// TwinCAT 3 PLC project HMISample
// ProgramVersion: 3.1.4022.1
// CompilerDefines: VISU_USEWSTRING
// libraries:
//   Tc2_ProfinetDiag, * (Beckhoff Automation GmbH)
//   Tc2_Standard, * (Beckhoff Automation GmbH)
//   Tc2_System, * (Beckhoff Automation GmbH)
//   Tc2_SystemCX, * (Beckhoff Automation GmbH)
//   Tc2_Utilities, * (Beckhoff Automation GmbH)
//   Tc3_Module, * (Beckhoff Automation GmbH)
//   VisuDialogs, * (System)
//   VisuSymbols,3.5.10.0,System
// project tree:
//   DUTs/ ST_EventDefinition.TcDUT, ST_EventHistoricalSimple.TcDUT, ST_EventHistoricalSimplePersistent.TcDUT
//   / GlobalTextList.TcGTLO, PlcTask.TcTTO, Visualization Manager.TcVMO (not stored), VISU_TASK.TcTTO
//   GVLs/ GVL_Checks.TcGVL, GVL_EHS.TcGVL, GVL_EHSP.TcGVL, GVL_HMI.TcGVL, ST_FileDialogParams.TcDUT
//   POUs/Checks/ CheckBounds.TcPOU, CheckDivDInt.TcPOU, CheckDivLInt.TcPOU, CheckDivLReal.TcPOU, CheckDivReal.TcPOU, CheckPointer.TcPOU, CheckRangeSigned.TcPOU, CheckRangeUnsigned.TcPOU
//   POUs/Events/Functions/ F_RESET_Event.TcPOU, F_SET_Event.TcPOU
//   POUs/Events/ P_Events.TcPOU, P_EventsDefinition.TcPOU, P_EventsHandling.TcPOU, P_EventsVisu.TcPOU
//   POUs/FBs/ FB_TaskInfo.TcPOU
//   POUs/ MAIN.TcPOU, P_CloseTcHmiExe.TcPOU, P_ControllerInfo.TcPOU, P_FileDialog.TcPOU, P_HmiControl.TcPOU, P_PersistentData.TcPOU, P_SystemInfo.TcPOU, P_Table.TcPOU, P_TaskInfo.TcPOU, P_UserControl.TcPOU
//   VISUs/Images/Buttons/ IP_Buttons.TcIPO (not stored)
//   VISUs/Images/ IP_Images.TcIPO (not stored)
//   VISUs/Internal/ Keypad.TcVIS, Numpad.TcVIS, PH_Bottom.TcVIS, PH_ControllerInfo.TcVIS, PH_Header.TcVIS, PH_Menu.TcVIS, PH_SystemInfo.TcVIS, PH_TaskInfo.TcVIS
//   VISUs/Menus/ V_FileDialog.TcVIS, V_Option6.TcVIS, V_Table.TcVIS, V_Trend.TcVIS, V_Option4.TcVIS, V_Option5.TcVIS
//   VISUs/ TL_Frames.TcTLO, TL_Lang.TcTLO, Visualization.TcVIS, V_EventsHistoricalSimple.TcVIS, V_Home.TcVIS, V_info.TcVIS, V_Settings.TcVIS, V_Users.TcVIS
// real-time tasks:
//   TASK PlcTask: cycle T#10ms, priority 20, ADS port 350
//   TASK VISU_TASK: cycle T#100000us, priority 30, ADS port 351

CONFIGURATION HMISample
    RESOURCE PLC ON TwinCAT3
        TASK PlcTask(INTERVAL := T#10ms, PRIORITY := 20);
        TASK VISU_TASK(INTERVAL := T#100000us, PRIORITY := 30);
        PROGRAM MAIN WITH PlcTask : MAIN;
        PROGRAM VisuElems_Visu_Prg WITH VISU_TASK : VisuElems.Visu_Prg;
    END_RESOURCE
END_CONFIGURATION

// ---- DUTs/ST_EventDefinition.TcDUT
//==================================================================================================
//							Beckhoff Automation Poland
//									23.05.2017
//	Struktura zawierajaca definicje zdarzenia
// 	v1.0	|| TC v 3.1.4020.32		|| - pierwsza wersja
//==================================================================================================
TYPE ST_EventDefinition :
STRUCT
	dwClass									: DWORD;
	dwParam									: DWORD;
	wsMessage								: WSTRING(80);
	bActive									: BOOL;	
END_STRUCT
END_TYPE

// ---- DUTs/ST_EventHistoricalSimple.TcDUT
//==================================================================================================
//							Beckhoff Automation Poland
//									23.05.2017
//	Struktura zawierajaca zdarzenie - pelne informacje, np. do wizualizacji
// 	v1.0	|| TC v 3.1.4020.32		|| - pierwsza wersja
//==================================================================================================
TYPE ST_EventHistoricalSimple :
STRUCT
	dwID									: DWORD;
	dwParam									: DWORD;
	dwClass									: DWORD;
	dtDateBegin								: DT;
	dtDateEnd								: DT;
	wsMessage								: WSTRING(80);
	dwColor									: UDINT;
END_STRUCT
END_TYPE

// ---- DUTs/ST_EventHistoricalSimplePersistent.TcDUT
//==================================================================================================
//							Beckhoff Automation Poland
//									23.05.2017
//	Struktura zawierajaca zane do przechowania zdarzenia w pamieci
// 	v1.0	|| TC v 3.1.4020.32		|| - pierwsza wersja
//==================================================================================================
TYPE ST_EventHistoricalSimplePersistent :
STRUCT
	dwID									: DWORD;
	dwParam									: DWORD;
	dwClass									: DWORD;
	dtDateBegin								: DT;
	dtDateEnd								: DT;
END_STRUCT
END_TYPE

// ---- GVLs/ST_FileDialogParams.TcDUT
TYPE ST_FileDialogParams :
STRUCT
	sDirectory 								: STRING(255);
	sFilter 								: STRING;
	sFileIn 								: STRING;
	sTitle 									: STRING;
	nRowCount								: INT;
	bBrowseDirectory						: BOOL;
	bTouch		 							: BOOL;
END_STRUCT
END_TYPE

// ---- GVLs/GVL_Checks.TcGVL
VAR_GLOBAL PERSISTENT
	dCheckBounds		: DINT;	(*Licznik przekroczen zakresu indexow, np. tablic*)
	dCheckDivDInt		: DINT;	(*Licznik prob dzielenia Dint przez 0*)
	dCheckDivLInt		: DINT; (*Licznik prob dzielenia LInt przez 0*)
	dCheckDivLReal		: DINT; (*Licznik prob dzielenia LREAL przez 0*)
	dCheckDivReal		: DINT; (*Licznik prob dzielenia REAL przez 0*)
	dCheckRangeSigned	: DINT;	(*Licznik przekroczen  liczby znakowej*)
	dCheckRangeUnsigned	: DINT; (*Licznik przekroczen  liczby bezznakowej*)
END_VAR

// ---- GVLs/GVL_EHS.TcGVL
//==================================================================================================
//							Beckhoff Automation Poland
//									23.05.2017
// 	v1.0	|| TC v 3.1.4020.32		|| - pierwsza wersja
//==================================================================================================
{attribute 'qualified_only'}
VAR_GLOBAL CONSTANT
	diEventsDefinition						: DINT 	:= 300;				// Rozmiar tablicy definicji zdarzen, powinna byc w zakresie 5..1000
	diNoOfEvents							: DINT 	:= 100;				// Rozmiar tablicy zdarzen historycznych, powinna byc w zakresie 5..1000
END_VAR
VAR_GLOBAL
	stActTime								: TIMESTRUCT;				// Aktualny czas sytemowy w formie struktury
	dtActTime								: DT;						// Aktualny czas sytemowy
	arrEventDefinition 						: ARRAY [1..GVL_EHS.diEventsDefinition] OF ST_EventDefinition;
	arrEventVisu							: ARRAY [1..GVL_EHS.diNoOfEvents] OF ST_EventHistoricalSimple;		// Pokazywane na wizualizacji - po filtracji
	dwLanguageId							: DWORD := 1033;			// Kod jezyka wyswietlania - Microsoft Locale ID Values
END_VAR

// ---- GVLs/GVL_EHSP.TcGVL
//==================================================================================================
//							Beckhoff Automation Poland
//									23.05.2017
// 	v1.0	|| TC v 3.1.4020.32		|| - pierwsza wersja
//==================================================================================================
{attribute 'qualified_only'}
VAR_GLOBAL PERSISTENT
	arrEvent								: ARRAY [1..GVL_EHS.diNoOfEvents] OF ST_EventHistoricalSimplePersistent;
END_VAR

// ---- GVLs/GVL_HMI.TcGVL
  
VAR_GLOBAL
	//numer strony
	iFrameNumber							: INT;
	//manu boczne
	bMain1									: BOOL;
	bMain2									: BOOL;
	udiFOntColor1							: UDINT;
	udiFOntColor2							: UDINT;
	bMenu									: BOOL;
	//alarmy
	arrEvents 						        : ARRAY [1..100] OF STRING;
	bReset									: BOOL;
	//test alarmów
	bAlarm									: BOOL;
	bWarning								: BOOL;
	bMessage								: BOOL;
	//jezyki
	iLang									: INT;
	//File dialog
	stFileDialogParams						: ST_FileDialogParams;
	bFileDialogOpen 						: BOOL := FALSE;
	//header
	wButton									: WORD; 				(* 	.0 - Menu,
																	.1 - Home,
																	.2 - Alarms,
																	.3 - Info,
																	.4 - Users,
																	.5 - Settings *)		
	wDeviceInfo								: WORD;		
								
END_VAR

// ---- POUs/MAIN.TcPOU
(*	| author		| Beckhoff Automation Poland	|	*)
(* 	-------------------------------------------------	*)
(*	| wersion		| 3.0							|	*)
(* 	-------------------------------------------------	*)
(*	| TC version	| 3.1.4024.7					| 	*)
(* 	-------------------------------------------------	*)
(*	| date			| 19.05.2020					|	*)
(* 	-------------------------------------------------	*)
(*	| description	| sample visu with navigation		
					  and frequently used functions	|  	*)
PROGRAM MAIN
VAR
END_VAR

P_HmiControl();
P_UserControl();
P_SystemInfo();
P_TaskInfo();
P_PersistentData();
P_Events();
P_FileDialog();
P_Table();
P_ControllerInfo();
P_CloseTcHmiExe();

END_PROGRAM

// ---- POUs/P_HmiControl.TcPOU
(*language & colors for visu*)
PROGRAM P_HmiControl
VAR

END_VAR

//zwijanie ruchomego menu po przelaczeniu na inne okno
IF NOT GVL_HMI.bMenu THEN
	GVL_HMI.bMain1:=FALSE;
	GVL_HMI.bMain2:=FALSE;
END_IF

IF GVL_HMI.bMain1 THEN
	GVL_HMI.udiFOntColor1:=16#FF404040;
ELSE 
	GVL_HMI.udiFOntColor1:=16#FFE5E5E5;
END_IF

IF GVL_HMI.bMain2 THEN
	GVL_HMI.udiFOntColor2:=16#FF404040;
ELSE 
	GVL_HMI.udiFOntColor2:=16#FFE5E5E5;
END_IF

IF GVL_HMI.iLang=0 THEN
	VisuElemsWinControls.CURRENTLANGUAGE:='EN';
ELSIF GVL_HMI.iLang=1 THEN
	VisuElemsWinControls.CURRENTLANGUAGE:='PL';
END_IF

END_PROGRAM

// ---- POUs/P_UserControl.TcPOU
(*program for controlling visu users from plc code*)
PROGRAM P_UserControl
VAR
	(*variables for tracking autologout time*)
	stTime 								: OTSTRUCT;
	sMin								: STRING;
	sSec								: STRING;
	sTime								: STRING;
	(*variables for listing existing users*)
	fbUserMng   						: VisuUserManagement.VisuUserMgmt;
   	stRet      							: VisuUserManagement.VUM_ReturnValues;
   	udiNumberOfUsers   					: UDINT;
   	dwUserDB         					: DWORD;
   	bUpdateUserList   					: BOOL;
   	aUserList         					: ARRAY[0..5] OF VisuUserManagement.VUM_User;
END_VAR

IF VisuElems.CurrentUseAutoLogoutTime THEN
	stTime 	:= TIME_TO_OTSTRUCT(VisuElems.CurrentRemainingAutoLogoutTime);
	sMin 	:= DWORD_TO_STRING(stTime.wMinute);
	sSec 	:= DWORD_TO_STRING(stTime.wSecond);
	sTime 	:= CONCAT(sMin, ':');
	sTime 	:= CONCAT(sTime, sSec);
ELSE
	sTime 	:= '';
END_IF

IF bUpdateUserList THEN
	bUpdateUserList:=FALSE;
   	dwUserDB := fbUserMng.GetUserDBAsCopy();
   	udiNumberOfUsers := fbUserMng.GetUserCount(dwUserDB);

 	stRet := fbUserMng.GetUsers(
                 dwUserDB:= dwUserDB, 
                 udiStartIndex:= 0, 
                 udiEndIndex:= udiNumberOfUsers-1, 
                 pArr:=  ADR(aUserList),
                 udiArrSize:= udiNumberOfUsers);
END_IF

END_PROGRAM

// ---- POUs/P_SystemInfo.TcPOU
//==================================================================================================
//							Beckhoff Automation Poland
//									P_SystemInfo
//									15.11.2016
//					Program odczytujący informacje o TC Runtime
// 
//	v1.1 	|| TC v 3.1.4020.14 	|| - Dodane wyjscia bOk, bWarning, bError
//	v1.0 	|| TC v 3.1.4020.0 		|| - Pierwsza wersja
//==================================================================================================
PROGRAM P_SystemInfo
VAR_INPUT
	bConfirm					: BOOL;					// Potwierdzenie bledu/ostrzezenia persistentow - blad/ostrzezenie nie znika, my usuwamy flage error lub warning
END_VAR
VAR_OUTPUT
	bOK							: BOOL;					// Zmienne wczytane prawidlowo
	bWarning					: BOOL;					// Zmienne wczytane z pliku zapasowego
	bError						: BOOL;					// Nie wczytano zmiennych
END_VAR
VAR
	sStartTime					: STRING;				// Przekonwertowany czas
END_VAR

//_AppInfo.ObjId; 			(* Object ID of the PLC project instance *)
//_AppInfo.TaskCnt;			(* The number of tasks in the actual runtime system *)
//_AppInfo.OnlineChangeCnt;	(* The number of online changes made since the last complete download. *)
//_AppInfo.Flags;				(* Reserved for future use *)
//_AppInfo.AdsPort; 			(* ADS port of PLC application *)
bOK							:= (_AppInfo.BootDataLoaded AND NOT _AppInfo.OldBootData) OR bConfirm;	(* PERSISTENT variables: LOADED (without error) *)
bWarning					:= _AppInfo.OldBootData AND NOT bConfirm;	(* PERSISTENT variables: INVALID (the back-up copy was loaded, since no valid data was present) *)
bError						:= NOT bOK AND NOT bWarning;
//_AppInfo.KeepOutputsOnBP;	(* The flag can be set to avoid that the outputs are zero-filled if a breakpoint is reached. The task keeps running. Only the execution of PLC code is interrupted. *)
//_AppInfo.TComSrvPtr;		(* Pointer to TcCOM Object Server *)
//_AppInfo.AppName;			(* TwinCAT generated name containing the port number. *)
//_AppInfo.ProjectName;		(* The name of the PLC project. *)
sStartTime					:= DELETE(DT_TO_STRING(_AppInfo.AppTimestamp),3,1);(* Date and time of application start *)
(*_AppInfo.BSODOccured;
_AppInfo.LicensesPending;
_AppInfo.ShutdownInProgress;*)

END_PROGRAM

// ---- POUs/P_TaskInfo.TcPOU
//==================================================================================================
//						Beckhoff Automation Poland
//							P_TaskInfo
//							15.11.2016
//
//				Program  odczytujący informacje o tasku
//
// 	v1.0 || TC v 3.1.4020.14 || - pierwsza wersja
//==================================================================================================
PROGRAM P_TaskInfo
VAR_OUTPUT
	bOK								: BOOL;	// Brak bledow i ostrzezen
	bWarning						: BOOL;	// Ostrzezenie - nie wystepuja w tym podprogramie - wystepuja dla zachowania spojnosci
	bError							: BOOL;	// Zbiorcza flaga bledow
	bReset							: BOOL; 
END_VAR
VAR
	fbTaskInfo						: FB_TaskInfo;
END_VAR

fbTaskInfo(bReset:=bReset , bError=> );
bError := fbTaskInfo.bError; // Dla jednego tasku. W przypadku wiekszej ilosci taskow trzeba dopisac reszte.

bOk := NOT bError;

END_PROGRAM

// ---- POUs/FBs/FB_TaskInfo.TcPOU
//==================================================================================================
//							Beckhoff Automation Poland
//							FB_TaskInfo
//							15.11.2016
//
//				Blok funkcyjny odczytujący informacje o tasku
//				Zapamiętuje maksymalne czasy wykonania oraz licznik przekroczeń
//
// 	v1.1 	|| TC v 3.1.4020.14 	|| - dodanie wyjsc
// 	v1.0 	|| TC v 3.1.4020.14 	|| - pierwsza wersja
//==================================================================================================
FUNCTION_BLOCK FB_TaskInfo
VAR_INPUT
	bReset					: BOOL;
END_VAR
VAR_OUTPUT
	bError					: BOOL;
END_VAR
VAR
	fbGetCurTaskIdx			: GETCURTASKINDEX;
	rLastExecTime			: REAL;
	rCycleTime				: REAL;
	uiPriority				: UINT;
	sTaskName				: STRING(63);
	bCycleTimeExceeded		: BOOL;
	rCycleCount				: REAL;
	rTotalTime				: REAL;
	rAverageCycleTime		: REAL;
	bResetVisu				: BOOL;
	byIndex					: BYTE;
END_VAR
VAR PERSISTENT
	udiCountExceedCycle		: UDINT; 						
	rMaxExecTime			: REAL;						
END_VAR

fbGetCurTaskIdx(index=>byIndex);

(*Odczyt czasu cyklu i ostatniego czasu wykonania*)
rCycleTime 					:= UDINT_TO_REAL(_TaskInfo[byIndex].CycleTime)/10000.0;
rLastExecTime 				:= UDINT_TO_REAL(_TaskInfo[byIndex].LastExecTime)/10000.0;
(*Zapamiętanie maksymalnego czasu wykonania*)
IF rLastExecTime > rMaxExecTime THEN 
	rMaxExecTime 			:= rLastExecTime;
END_IF

uiPriority					:= _TaskInfo[byIndex].Priority;
sTaskName					:= _TaskInfo[byIndex].TaskName;
bCycleTimeExceeded			:= _TaskInfo[byIndex].CycleTimeExceeded;
bError 						:= bCycleTimeExceeded; // Blad gdy czas cyklu przekroczony

(*Licznik przekroczeń czasu cyklu*)
IF _TaskInfo[byIndex].CycleTimeExceeded  THEN 
	udiCountExceedCycle 	:= udiCountExceedCycle + 1; 
END_IF
rCycleCount 				:= rCycleCount + 1;
rTotalTime 					:= rLastExecTime + rTotalTime;
rAverageCycleTime 			:= rTotalTime / rCycleCount;

(*Reset wyliczanych wartości*)
IF bReset OR bResetVisu THEN
	udiCountExceedCycle 	:= 0;
	rMaxExecTime 			:= 0;
	rTotalTime 				:= 0;
	rCycleCount 			:= 0;
	rAverageCycleTime 		:= 0;
	bReset 					:= FALSE;
END_IF

END_FUNCTION_BLOCK

// ---- POUs/P_PersistentData.TcPOU
PROGRAM P_PersistentData
VAR
	writepersistent							: WRITEPERSISTENTDATA;
	bWrite									: BOOL;
	udiErrID								: UDINT;
END_VAR
VAR PERSISTENT
	iInt1									: INT:=10;
END_VAR

writepersistent(PORT := 851, START := bWrite); // WRITEPERSISTENTDATA
udiErrID := writepersistent.ERRID;

END_PROGRAM

// ---- POUs/Events/P_Events.TcPOU
//==================================================================================================
//							Beckhoff Automation Poland
//									23.05.2017
//	Program obslugujacy proste alarmy historyczne.
//	W opcjach wizualizacji trzeba wybrac use uniceode strings i use current visu variable
// 	v1.0	|| TC v 3.1.4020.32		|| - pierwsza wersja
//==================================================================================================
PROGRAM P_Events
VAR
	fbLocalSystemTime						: FB_LocalSystemTime;
	bEventTableSizeError					: BOOL;					// Niewlasciwy rozmiar tablicy zdarzen - sprawdz GVL_EHS.diNoOfEvents
	bEventDefinitionSizeError				: BOOL;					// Niewlasciwy rozmiar tablicy zdarzen - sprawdz GVL_EHS.diEventsDefinition
END_VAR

fbLocalSystemTime(bEnable:= TRUE, systemTime=> GVL_EHS.stActTime);
GVL_EHS.dtActTime 							:= SYSTEMTIME_TO_DT(GVL_EHS.stActTime);

P_EventsDefinition ();

bEventDefinitionSizeError 					:= GVL_EHS.diEventsDefinition < 5 OR GVL_EHS.diEventsDefinition > 1000;
bEventTableSizeError 						:= GVL_EHS.diNoOfEvents < 5 OR GVL_EHS.diNoOfEvents > 1000;

IF NOT bEventDefinitionSizeError AND NOT bEventTableSizeError THEN
	IF fbLocalSystemTime.bValid THEN
		P_EventsHandling();
	END_IF
	// Visu i filtry
	P_EventsVisu();	
END_IF

END_PROGRAM

// ---- POUs/Events/P_EventsDefinition.TcPOU
//==================================================================================================
//							Beckhoff Automation Poland
//									23.05.2017
//	Program definiujacy zdarzenia - musi byc dostosowany do aplikacji
//	W pierwszym cyklu definiowane sa klasy
//	Zmiana jezyka na zdarzenie i w pierwszym cyklu
//	Wykrywanie aktywnosci zdarzenia i parametru - cykliczne
// 	v1.0	|| TC v 3.1.4020.32		|| - pierwsza wersja
//==================================================================================================
PROGRAM P_EventsDefinition
VAR
	bFirstCycle 							: BOOL := TRUE;
	dwPreviousLanguageID					: DWORD;
	i										: INT;
END_VAR

// Class
IF bFirstCycle THEN
	ACT_ClassDefinition();
	bFirstCycle 							:= FALSE;
END_IF

// Language
ACT_Language();

// Active
ACT_Active();

ACTION ACT_1033_US:
// Fatal Error
GVL_EHS.arrEventDefinition[1].wsMessage	 	:= "Error01";

// Warning
GVL_EHS.arrEventDefinition[101].wsMessage 	:= "Warning01";

// Message
GVL_EHS.arrEventDefinition[201].wsMessage 	:= "Message01";
END_ACTION

ACTION ACT_1045_PL:
//
END_ACTION

ACTION ACT_Active:
GVL_EHS.arrEventDefinition[1].bActive:= GVL_HMI.bAlarm;
GVL_EHS.arrEventDefinition[101].bActive:=GVL_HMI.bWarning;
GVL_EHS.arrEventDefinition[201].bActive:=GVL_HMI.bMessage;
END_ACTION

ACTION ACT_ClassDefinition:
FOR i := 1 TO 100 DO
	// Error - [1..100] - Class 0
	GVL_EHS.arrEventDefinition[i].dwClass := 0;
	// Warning - [101..200] - Class 1
	GVL_EHS.arrEventDefinition[100+i].dwClass := 1;
	// Message - [201..300] - Class 2
	GVL_EHS.arrEventDefinition[200+i].dwClass := 2;
END_FOR
END_ACTION

ACTION ACT_Language:
// Wybor jezyka
IF dwPreviousLanguageID <> GVL_EHS.dwLanguageId THEN
	CASE GVL_EHS.dwLanguageId OF
		
		1033:	// United States
			ACT_1033_US();
			
		1045:	// Polish
			ACT_1045_PL();
	
	ELSE	// Default Polish
		
			ACT_1045_PL();
	END_CASE
END_IF

dwPreviousLanguageID := GVL_EHS.dwLanguageId;
END_ACTION

END_PROGRAM

// ---- POUs/Events/P_EventsHandling.TcPOU
//==================================================================================================
//							Beckhoff Automation Poland
//									23.05.2017
//	Program obslugujacy zdarzenia historyczne - edycji podlega tylko tRefreshTime i bRealTime
// 	v1.0	|| TC v 3.1.4020.32		|| - pierwsza wersja
//==================================================================================================
PROGRAM P_EventsHandling
VAR
	bRealTime								: BOOL := TRUE;		// Odswiezanie ciagle - zmieniamy na FALSE tylko gdy jest duze obciazenie CPU
																// Zmiana na FLASE powoduje odfiltrowanie alarmow zgodnie z czasem tRefreshTime
	tonRefresh								: TON;				// Timer odswiezenia
	tRefreshTime							: TIME := T#1S;		// Czestotliwosc odswiezania - im dluzszy szac tym wieksze ryzyko niezauwazenia wystapienia alarmu
	bInitialized							: BOOL;				// Flaga inicjalizacji
	i										: DINT;				// Iterator petli
	// Tablice wykrycia poczatku/konca zdarzenia
	arrSet									: ARRAY [1..GVL_EHS.diEventsDefinition] OF R_TRIG;
	arrReset								: ARRAY [1..GVL_EHS.diEventsDefinition] OF F_TRIG;
END_VAR

// Inicjalizacja - po uruchomieniu znajdz niezakonczone alarmy i dodaj aktualny czas jako zakonczenie
IF NOT bInitialized THEN
	FOR i := 1 TO GVL_EHS.diEventsDefinition DO
		F_RESET_Event(dwID:= i, dtActTime:= GVL_EHS.dtActTime);
	END_FOR	
	bInitialized 							:= TRUE;
END_IF

// Timer odswiezania
tonRefresh(IN:= NOT tonRefresh.Q, PT:= tRefreshTime, Q=> , ET=> );

IF bRealTime OR tonRefresh.Q THEN
	FOR i := 1 TO GVL_EHS.diEventsDefinition DO
		// Wykrycie pojawienia sie zdarzenia - ustawienie flagi na 1 cykl i dodanie na poczatek listy
		arrSet[i](CLK:= GVL_EHS.arrEventDefinition[i].bActive);
		IF arrSet[i].Q THEN
			F_SET_Event(dwID:= i, stEventDefinition:= GVL_EHS.arrEventDefinition[i], dtActTime:= GVL_EHS.dtActTime);
		END_IF
		// Wykrycie zakonczenia zdarzenia - ustawienie flagi na 1 cykl i dodanie daty zakonczenia
		arrReset[i](CLK:= GVL_EHS.arrEventDefinition[i].bActive);
		IF arrReset[i].Q THEN
			F_RESET_Event(dwID:= i, dtActTime:= GVL_EHS.dtActTime);
		END_IF
	END_FOR	
END_IF

END_PROGRAM

// ---- POUs/Events/Functions/F_RESET_Event.TcPOU
FUNCTION F_RESET_Event : BOOL
VAR_INPUT
	dwID									: DWORD;
	dtActTime								: DT;
END_VAR
VAR
	i										: DINT;
END_VAR

// Znajdz i wstaw date zakonczenia
FOR i := 1 TO GVL_EHS.diNoOfEvents DO
	IF 	GVL_EHSP.arrEvent[i].dwID = dwID THEN
		GVL_EHSP.arrEvent[i].dtDateEnd		:= dtActTime;
		EXIT;
	END_IF
END_FOR

END_FUNCTION

// ---- POUs/Events/Functions/F_SET_Event.TcPOU
FUNCTION F_SET_Event : BOOL
VAR_INPUT
	dwID									: DWORD;
	stEventDefinition						: ST_EventDefinition;
	dtActTime								: DT;
END_VAR
VAR
	i										: DINT;
END_VAR

// Przesun elemety tablicy
FOR i := 0 TO GVL_EHS.diNoOfEvents-2 DO
	GVL_EHSP.arrEvent[GVL_EHS.diNoOfEvents-i] := GVL_EHSP.arrEvent[GVL_EHS.diNoOfEvents-i-1];
END_FOR
// Dodaj nowy
GVL_EHSP.arrEvent[1].dwID					:= dwID;
GVL_EHSP.arrEvent[1].dtDateBegin 			:= dtActTime;
GVL_EHSP.arrEvent[1].dtDateEnd	 			:= DT#1970-1-1-0:0:0;
GVL_EHSP.arrEvent[1].dwParam 				:= stEventDefinition.dwParam;
GVL_EHSP.arrEvent[1].dwClass 				:= stEventDefinition.dwClass;

END_FUNCTION

// ---- POUs/Events/P_EventsVisu.TcPOU
//==================================================================================================
//							Beckhoff Automation Poland
//									23.05.2017
//	Program obslugujacy wizualizacje VISU_EventsHistoricalSimple
//	Mozliwe filtrowanie alamow. Czestotliwosc odswiezania wplywa tylko na wyswietlanie
// 	v1.0	|| TC v 3.1.4020.32		|| - pierwsza wersja
//==================================================================================================
PROGRAM P_EventsVisu
VAR
	i										: DINT;				// Iterator tablicy przechowywanej w pamieci
	j										: DINT;				// Iterator tablicy wyswietlanej
	bActiveWindow							: BOOL := TRUE;		// Flaga wysietlania okna - tylko wtedy odswiezamy tablice wyswietlana
	rtPageChange							: R_TRIG;			// Wykrycie przelaczenia strony
	tonRefresh								: TON;
	tRefreshTime							: TIME := T#50MS;	// Czestotliwosc odswiezania strony
	//========================= Filtry =========================
	bRemoveFromList							: BOOL; 			// Flaga pomocnicza dla filtrow - decyduje czy element ma byc dodany na wizualizacje
	// Flagi wykonywalnosci
	bFilterID								: BOOL;
	bFilterClass							: BOOL;
	bFilterActiveOnly						: BOOL;
	// Parametry
	dwFilterID								: DWORD;	
	dwFilterClass							: DWORD;
END_VAR

bActiveWindow := TRUE;//VisuElems.CURRENTVISU = 'VISU_EventsHistoricalSimple';						// Flaga wysietlania okna
rtPageChange(CLK:= bActiveWindow, Q=> );													// Wykrycie zmiany strony - jednorazowo inicjalizacja
tonRefresh(IN:= bActiveWindow AND NOT tonRefresh.Q, PT:= tRefreshTime, Q=> , ET=> );		// Timer odswiezania

IF  rtPageChange.Q OR tonRefresh.Q THEN
	// Czyszczenie tablicy
	MEMSET(ADR(GVL_EHS.arrEventVisu),0,SIZEOF(GVL_EHS.arrEventVisu));
	j := 1;
	// Filters
	FOR i := 1 TO GVL_EHS.diNoOfEvents DO
		bRemoveFromList 								:= FALSE;
		// Jesli jest element
		IF GVL_EHSP.arrEvent[i].dwID <> 0 THEN
			bRemoveFromList								:= bFilterID AND dwFilterID <> GVL_EHSP.arrEvent[i].dwID;
			bRemoveFromList								:= bRemoveFromList OR (bFilterClass AND dwFilterClass <> GVL_EHSP.arrEvent[i].dwClass);
//			bRemoveFromList								:= bRemoveFromList OR (bFilterBeginTimeFrom AND GVL_EHSP.arrEvent[i].dtDateBegin <= dtFilterBeginTimeFrom);
//			bRemoveFromList								:= bRemoveFromList OR (bFilterBeginTimeTo AND GVL_EHSP.arrEvent[i].dtDateBegin >= dtFilterBeginTimeTo);
//			bRemoveFromList								:= bRemoveFromList OR (bFilterEndTimeFrom AND GVL_EHSP.arrEvent[i].dtDateEnd <= dtFilterEndTimeFrom);
//			bRemoveFromList								:= bRemoveFromList OR (bFilterEndTimeTo AND GVL_EHSP.arrEvent[i].dtDateEnd >= dtFilterEndTimeTo);
			bRemoveFromList								:= bRemoveFromList OR (bFilterActiveOnly AND DT#1970-1-1-0:0:0 <> GVL_EHSP.arrEvent[i].dtDateEnd);
			// Analogicznie dodajemy inne filtry jesli jest taka potrzeba
			// Jesli element nie zostal usuniety przez filtr to dodajemy go do tablicy alarmow wyswietlanych
			IF NOT bRemoveFromList THEN
				GVL_EHS.arrEventVisu[j].dwID 			:= GVL_EHSP.arrEvent[i].dwID;
				GVL_EHS.arrEventVisu[j].dwClass 		:= GVL_EHSP.arrEvent[i].dwClass;
				GVL_EHS.arrEventVisu[j].wsMessage		:= GVL_EHS.arrEventDefinition[GVL_EHSP.arrEvent[i].dwID].wsMessage;
				GVL_EHS.arrEventVisu[j].dwParam 		:= GVL_EHSP.arrEvent[i].dwParam;
				GVL_EHS.arrEventVisu[j].dtDateBegin 	:= GVL_EHSP.arrEvent[i].dtDateBegin;
				GVL_EHS.arrEventVisu[j].dtDateEnd 		:= GVL_EHSP.arrEvent[i].dtDateEnd;
				IF GVL_EHS.arrEventVisu[j].dwClass=0 THEN
					GVL_EHS.arrEventVisu[j].dwColor:=16#FFFF0000;
				ELSIF GVL_EHS.arrEventVisu[j].dwClass=1 THEN
					GVL_EHS.arrEventVisu[j].dwColor:=16#FFF3F24A;
				ELSIF GVL_EHS.arrEventVisu[j].dwClass=2 THEN
					GVL_EHS.arrEventVisu[j].dwColor:=16#FF4E9640;
				END_IF
				j := j + 1;
			END_IF 
		END_IF
	END_FOR
END_IF

END_PROGRAM

// ---- POUs/P_FileDialog.TcPOU
(*program for setting parameters for FileOpenSae visualization dialog*)
PROGRAM P_FileDialog
VAR
	fbFileList                              : Visu_FbFileListProvider; 
	sSelectedDirectory						: STRING;
	sSelectedFileName						: STRING;
	iCount									: INT;
	bOpen 									: BOOL;
	sDir									: STRING(255):='C:\';
	bFile									: BOOL:=TRUE;
END_VAR

IF bFile OR bOpen THEN
	fbFileList.Initialize(
                        stDirectory:= sDir, 
                        stFilter:='Text Files(*.txt)|*.txt' , 
                        stFileIn:='', 
                        stTitle:= 'Dialog file open', 
                        iRowCount:=10 , 
                        bBrowseDirectory:= TRUE, 
                        bTouch:=FALSE ); 
	bFile:=FALSE;
END_IF
					
 
sSelectedDirectory:=fbFileList.GetSelectedDirectory();
sSelectedFileName:=fbFileList.GetSelectedFileName();
iCount:=fbFileList.Count;

END_PROGRAM

// ---- POUs/P_Table.TcPOU
(*program for displaying data in Histogram visualization element*)
PROGRAM P_Table
VAR
	arrTable								: ARRAY [1..10,1..10] OF INT;
	i										: INT;
	j										: INT;
	a										: INT;
	bInit									: BOOL:=TRUE;
	iValue									: INT;
	iColumn									: INT:=1;
	iLine									: INT:=1;
	iSetValue								: INT;
	bSetNewValue							: BOOL;
	
	arrHistogram							: ARRAY [1..20] OF INT := [1, 2, 20, 15, 10, 6, 7, 8, 11, 10, 11, 12, 3(5), 6, 10, 18, 19, 20];	
	i1										: INT;
	iTemp									: INT;
	bRotate									: BOOL;
END_VAR

i:=0;
j:=0;
a:=1;
IF bInit THEN
	FOR i:=1 TO 10 DO
		FOR j:=1 TO 10 DO
			arrTable[i,j]:=a;
			a:=a+1;
		 END_FOR
	END_FOR
	bInit:=FALSE;
END_IF
iValue:=arrTable[iColumn,iLine];
IF bSetNewValue THEN
	arrTable[iColumn,iLine]:=iSetValue;
END_IF


IF bRotate THEN
	iTemp:=arrHistogram[1];
	FOR i1:=1 TO 19 DO
		arrHistogram[i1]:=arrHistogram[i1+1];
	END_FOR
	arrHistogram[20]:=iTemp;
END_IF

END_PROGRAM

// ---- POUs/P_ControllerInfo.TcPOU
(*program reading information about the controller *)
PROGRAM P_ControllerInfo
VAR
	fbCxGetDeviceIdentification				: FB_CxGetDeviceIdentification;
	stDevIdent 								: ST_CxDeviceIdentification;
	arrDevIdent								: ARRAY [0..1, 1..16] OF STRING(23) := [	'Target type:', 'Hardware Model:', 'Hardware Serial No:', 'Hardware Version:', 
														'Hardware Date:', 'Hardware CPU:', 'Image Device:', 'Image Version:', 'Image Level:', 
														'Image OS Name:', 'Image OS Version:', 'TwinCAT Version:', 'TwinCAT Revision:', 
														'TwinCAT Build:', 'TwinCAT Level:', 'AMS NET ID:', 16('')];
	iSelectedRow							: INT:=1;
END_VAR

fbCxGetDeviceIdentification(bExecute:=TRUE ,	stDevIdent=>stDevIdent);
IF NOT fbCxGetDeviceIdentification.bBusy AND NOT fbCxGetDeviceIdentification.bError THEN
	
	
	// for visu table
	arrDevIdent[1,1] := stDevIdent.strTargetType;
	arrDevIdent[1,2] := stDevIdent.strHardwareModel;
	arrDevIdent[1,3] := stDevIdent.strHardwareSerialNo;
	arrDevIdent[1,4] := stDevIdent.strHardwareVersion;
	arrDevIdent[1,5] := stDevIdent.strHardwareDate;
	arrDevIdent[1,6] := stDevIdent.strHardwareCPU;
	arrDevIdent[1,7] := stDevIdent.strImageDevice;
	arrDevIdent[1,8] := stDevIdent.strImageVersion;
	arrDevIdent[1,9] := stDevIdent.strImageLevel;
	arrDevIdent[1,10] := stDevIdent.strImageOsName;
	arrDevIdent[1,11] := stDevIdent.strImageOsVersion;
	arrDevIdent[1,12] := stDevIdent.strTwinCATVersion;
	arrDevIdent[1,13] := stDevIdent.strTwinCATRevision;
	arrDevIdent[1,14] := stDevIdent.strTwinCATBuild;
	arrDevIdent[1,15] := stDevIdent.strTwinCATLevel;
	arrDevIdent[1,16] := stDevIdent.strAmsNetId;
END_IF

END_PROGRAM

// ---- POUs/P_CloseTcHmiExe.TcPOU
PROGRAM P_CloseTcHmiExe
(*program for closing the visualization (terminates Tc3PlcHMi.exe process), 
 to terminate process, set bKillProcess var to TRUE*)
VAR
	bKillProcess							: BOOL;
	ntKillProcess							: NT_StartProcess;
END_VAR

ntKillProcess(
	NETID:='' ,
	PATHSTR:='C:\WINDOWS\system32\taskkill.exe' ,
	DIRNAME:='' , 
	COMNDLINE:='/t /f /IM Tc3PlcHmi.exe' , 
	START:= bKillProcess,
	ERRID=> );
bKillProcess := FALSE;

END_PROGRAM

// ---- POUs/Checks/CheckBounds.TcPOU
// Implicitly generated code : DO NOT EDIT
FUNCTION CheckBounds : DINT
VAR_INPUT
	index, lower, upper: DINT;
END_VAR

// Implicitly generated code : Only an Implementation suggestion
IF  index < lower THEN
	CheckBounds := lower;
	dCheckBounds := dCheckBounds + 1;
ELSIF  index > upper THEN
	CheckBounds := upper;
	dCheckBounds := dCheckBounds + 1;
ELSE  
	CheckBounds := index;
END_IF

END_FUNCTION

// ---- POUs/Checks/CheckDivDInt.TcPOU
// Implicitly generated code : DO NOT EDIT
FUNCTION CheckDivDInt : DINT
VAR_INPUT
	divisor:DINT;
END_VAR

// Implicitly generated code : Only an Implementation suggestion
IF divisor = 0 THEN
	CheckDivDInt:=1;
	dCheckDivDInt := dCheckDivDInt + 1;
ELSE
	CheckDivDInt:=divisor;
END_IF;

END_FUNCTION

// ---- POUs/Checks/CheckDivLInt.TcPOU
// Implicitly generated code : DO NOT EDIT
FUNCTION CheckDivLInt : LINT
VAR_INPUT
	divisor:LINT;
END_VAR

// Implicitly generated code : Only an Implementation suggestion
IF divisor = 0 THEN
	CheckDivLInt:=1;
	dCheckDivLInt := dCheckDivLInt + 1;
ELSE
	CheckDivLInt:=divisor;
END_IF;

END_FUNCTION

// ---- POUs/Checks/CheckDivLReal.TcPOU
// Implicitly generated code : DO NOT EDIT
FUNCTION CheckDivLReal : LREAL
VAR_INPUT
	divisor:LREAL;
END_VAR

// Implicitly generated code : Only an Implementation suggestion
IF divisor = 0 THEN
	CheckDivLReal:=1;
	dCheckDivLReal := dCheckDivLReal + 1;
ELSE
	CheckDivLReal:=divisor;
END_IF;

END_FUNCTION

// ---- POUs/Checks/CheckDivReal.TcPOU
// Implicitly generated code : DO NOT EDIT
FUNCTION CheckDivReal : REAL
VAR_INPUT
	divisor:REAL;
END_VAR

// Implicitly generated code : Only an Implementation suggestion
IF divisor = 0 THEN
	CheckDivReal:=1;
	dCheckDivReal := dCheckDivReal + 1;
ELSE
	CheckDivReal:=divisor;
END_IF;

END_FUNCTION

// ---- POUs/Checks/CheckPointer.TcPOU
// Implicitly generated code : DO NOT EDIT
FUNCTION CheckPointer : POINTER TO BYTE
VAR_INPUT 
	ptToTest : POINTER TO BYTE; // Destination address of the pointer
	iSize : DINT;		        // Size of the type the pointer points to. (e.g: 20 for POINTER TO ARRAY [0..9] OF INT) 
	iGran : DINT;		        // Granularity of the pointer access. This is the size of the biggest non-structured data type in the type the pointer points to. (e.g: 2 for POINTER TO ARRAY [0..9] OF INT)
	bWrite: BOOL;		        // Indicates read or write Access. TRUE = write access.
END_VAR

// No standard way of implementation. Fill your own code here
CheckPointer := ptToTest;

END_FUNCTION

// ---- POUs/Checks/CheckRangeSigned.TcPOU
// Implicitly generated code : DO NOT EDIT
FUNCTION CheckRangeSigned : DINT
VAR_INPUT
	value, lower, upper: DINT;
END_VAR

// Implicitly generated code : Only an Implementation suggestion
IF (value < lower) THEN
	CheckRangeSigned := lower;
	dCheckRangeSigned := dCheckRangeSigned + 1;
ELSIF(value > upper) THEN
	CheckRangeSigned := upper;
	dCheckRangeSigned := dCheckRangeSigned + 1;
ELSE
	CheckRangeSigned := value;
END_IF

END_FUNCTION

// ---- POUs/Checks/CheckRangeUnsigned.TcPOU
// Implicitly generated code : DO NOT EDIT
FUNCTION CheckRangeUnsigned : UDINT
VAR_INPUT
	value, lower, upper: UDINT;
END_VAR

// Implicitly generated code : Only an Implementation suggestion
IF (value < lower) THEN
	CheckRangeUnsigned := lower;
	dCheckRangeUnsigned := dCheckRangeUnsigned + 1;
ELSIF(value > upper) THEN
	CheckRangeUnsigned := upper;
	dCheckRangeUnsigned := dCheckRangeUnsigned + 1;
ELSE
	CheckRangeUnsigned := value;
END_IF

END_FUNCTION

// ---- GlobalTextList.TcGTLO
TEXTLIST GlobalTextList
  791 = '  '
  136 = '   Czas cyklu' | EN\: 'Cycle Time' | PL: 'Czas cyklu'
  149 = '  Przekroczony cykl' | EN\: 'Exceeded cycle ' | PL: 'Przekroczony cykl'
  969 = '  Reamining time: %s' | EN\: 'Remaining time: %s' | PL: 'Pozostały czas: %s'
  460 = '  Stan zmiennych persistent' | EN\: 'Persistent variables' | PL: 'Stan zmiennych persistent'
  517 = '  User group: %s' | EN\: 'User group: %s' | PL: 'Grupa użytkowników: %s'
  589 = '  User Name: %s' | EN\: 'User name: %s' | PL: 'Nazwa użytkownika: %s'
  340 = '!' | EN\: '!' | PL: '!'
  343 = '"' | EN\: '"' | PL: '"'
  973 = '#' | EN\: '#' | PL: '#'
  346 = '$' | EN\: '$' | PL: '$'
  350 = '%' | EN\: '%' | PL: '%'
  425 = '%.3f' | EN\: '%.3f' | PL: '%.3f'
  1614 = '%d' | EN\: '%d' | PL: '%d'
  703 = '%s' | EN\: '%s' | PL: '%s'
  214 = '%t[dd/MM/yyyy]' | EN\: '%t[dd/MM/yyyy]' | PL: '%t[dd/MM/yyyy]'
  213 = '%t[HH:mm:ss]' | EN\: '%t[HH:mm:ss]' | PL: '%t[HH:mm:ss]'
  353 = '&' | EN\: '&' | PL: '&'
  477 = "'" | EN\: "'" | PL: "'"
  356 = '(' | EN\: '(' | PL: '('
  360 = ')' | EN\: ')' | PL: ')'
  330 = '*' | EN\: '*' | PL: '*'
  328 = '+' | EN\: '+' | PL: '+'
  284 = '+/-' | EN\: '+/-' | PL: '+/-'
  480 = ',' | EN\: ',' | PL: ','
  448 = '-' | EN\: '-' | PL: '-'
  484 = '.' | EN\: '.' | PL: '.'
  488 = '/' | EN\: '/' | PL: '/'
  445 = '0' | EN\: '0' | PL: '0'
  1182 = '05-500 Piaseczno' | EN\: '05-500 Piaseczno' | PL: '05-500 Piaseczno'
  600 = '1' | EN\: '1' | PL: '1'
  1325 = '10' | EN\: '10' | PL: '10'
  606 = '2' | EN\: '2' | PL: '2'
  421 = '3' | EN\: '3' | PL: '3'
  423 = '4' | EN\: '4' | PL: '4'
  894 = '48 22 / 7 50 47 00' | EN\: '48 22 / 7 50 47 00' | PL: '48 22 / 7 50 47 00'
  427 = '5' | EN\: '5' | PL: '5'
  430 = '6' | EN\: '6' | PL: '6'
  434 = '7' | EN\: '7' | PL: '7'
  437 = '8' | EN\: '8' | PL: '8'
  441 = '9' | EN\: '9' | PL: '9'
  788 = ':' | EN\: ':' | PL: ':'
  473 = ';' | EN\: ';' | PL: ';'
  773 = '<' | EN\: '<' | PL: '<'
  452 = '=' | EN\: '=' | PL: '='
  774 = '>' | EN\: '>' | PL: '>'
  298 = '>>' | EN\: '>>' | PL: '>>'
  363 = '?' | EN\: '?' | PL: '?'
  974 = '@' | EN\: '@' | PL: '@'
  218 = 'A' | EN\: 'A' | PL: 'A'
  790 = 'a' | EN\: 'a' | PL: 'a'
  1771 = 'Active Only' | EN\: 'Active onlny' | PL: 'Tylko aktywne'
  578 = 'Admin' | EN\: 'Admin' | PL: 'Admin'
  1640 = 'Alarm'
  783 = 'b' | EN\: 'b' | PL: 'b'
  784 = 'B' | EN\: 'B' | PL: 'B'
  282 = 'Back' | EN\: 'Back' | PL: 'Back'
  417 = 'Backspace' | EN\: 'Backspace' | PL: 'Backspace'
  2094 = 'Beckhoff Automation Poland ' | EN\: 'Beckhoff Automation Polad' | PL: 'Beckhoff Automation Polad'
  957 = 'Błąd' | EN\: 'Error' | PL: 'Błąd'
  779 = 'c' | EN\: 'c' | PL: 'c'
  780 = 'C' | EN\: 'C' | PL: 'C'
  57 = 'Change Password' | EN\: 'Change Password' | PL: 'Zmień hasło'
  416 = 'Clear' | EN\: 'Clear' | PL: 'Clear'
  1188 = 'Close' | EN\: 'Close' | PL: 'Zamknij'
  1928 = 'Current User: %s' | EN\: 'Current User: %s' | PL: 'Użytkownik: %s'
  424 = 'Czas cyklu' | EN\: 'Cycle time' | PL: 'Czas cyklu'
  315 = 'Czas rozpoczęcia pracy: %s' | EN\: 'Work started : %s' | PL: 'Czas rozpoczęcia pracy: %s'
  610 = 'd' | EN\: 'd' | PL: 'd'
  611 = 'D' | EN\: 'D' | PL: 'D'
  1530 = 'Device Info' | EN\: 'Device Info' | PL: 'Device Info'
  492 = 'Directory and File Name' | EN\: 'Directory and file name' | PL: 'Ścieżka i nazwa pliku'
  490 = 'Directory to Open' | EN\: 'Directory to open' | PL: 'Ścieżka'
  979 = 'e' | EN\: 'e' | PL: 'e'
  980 = 'E' | EN\: 'E' | PL: 'E'
  415 = 'ESC' | EN\: 'ESC' | PL: 'ESC'
  612 = 'f' | EN\: 'f' | PL: 'f'
  613 = 'F' | EN\: 'F' | PL: 'F'
  288 = 'File Dialog' | EN\: 'File Dialog' | PL: 'Dialog plików'
  495 = 'File Name' | EN\: 'File Name' | PL: 'Nazwa pliku'
  614 = 'g' | EN\: 'g' | PL: 'g'
  615 = 'G' | EN\: 'G' | PL: 'G'
  217 = 'H' | EN\: 'H' | PL: 'H'
  616 = 'h' | EN\: 'h' | PL: 'h'
  219 = 'I' | EN\: 'I' | PL: 'I'
  988 = 'i' | EN\: 'i' | PL: 'i'
  1588 = 'Index: %d' | EN\: 'Index: %d' | PL: 'Index: %d'
  1562 = 'Info task' | EN\: 'Info task' | PL: 'Info task'
  1571 = 'Informacje o  tasku' | EN\: 'Task Info' | PL: 'Informacje o tasku'
  1597 = 'Informacje o przekroczonym cyklu' | EN\: 'Cycle exceeded' | PL: 'Informacje o przekroczonym cyklu'
  617 = 'j' | EN\: 'j' | PL: 'j'
  618 = 'J' | EN\: 'J' | PL: 'J'
  619 = 'k' | EN\: 'k' | PL: 'k'
  970 = 'K' | EN\: 'K' | PL: 'K'
  303 = 'Kolumna: %d' | EN\: 'Column: %d' | PL: 'Kolumna: %d'
  971 = 'l' | EN\: 'l' | PL: 'l'
  972 = 'L' | EN\: 'L' | PL: 'L'
  546 = 'Language:' | EN\: 'Language:' | PL: 'Język:'
  311 = 'Liczba tasków: %d' | EN\: 'Task count:  %d' | PL: 'Liczba tasków: %d'
  313 = 'Liczba zmian online: %d' | EN\: 'Online changes: %d' | PL: 'Liczba zmian online: %d'
  1622 = 'Licznik przekroczeń cyklu' | EN\: 'Exceeded cycle counter' | PL: 'Licznik przekroczeń cyklu'
  482 = 'Login' | EN\: 'Login' | PL: 'Login'
  77 = 'Logout' | EN\: 'Logout' | PL: 'Logout'
  216 = 'M' | EN\: 'M' | PL: 'M'
  787 = 'm' | EN\: 'm' | PL: 'm'
  826 = 'Main1' | EN\: 'Main1' | PL: 'Main1'
  557 = 'Main2' | EN\: 'Main2' | PL: 'Main2'
  706 = 'Maintenance' | EN\: 'Maintenance' | PL: 'Maintenance'
  105 = 'Max. czas cyklu' | EN\: 'Max. cycle time' | PL: 'Max. czas cyklu'
  590 = 'Max:' | EN\: 'Max:' | PL: 'Max:'
  475 = 'Message'
  585 = 'Min:' | EN\: 'Min:' | PL: 'Min:'
  785 = 'n' | EN\: 'n' | PL: 'n'
  786 = 'N' | EN\: 'N' | PL: 'N'
  309 = 'Nazwa projektu: %s' | EN\: 'Project name: %s' | PL: 'Nazwa projektu: %s'
  1579 = 'Nazwa tasku: %s' | EN\: 'Task name: %s' | PL: 'Nazwa tasku: %s'
  422 = 'NIE' | EN\: 'No' | PL: 'NIE'
  881 = 'None' | EN\: 'None' | PL: 'None'
  1107 = 'Nowa wartość: %d' | EN\: 'New value: %d' | PL: 'Nowa wartość: %d'
  989 = 'o' | EN\: 'o' | PL: 'o'
  990 = 'O' | EN\: 'O' | PL: 'O'
  414 = 'OK' | EN\: 'OK' | PL: 'OK'
  1097 = 'Open Dialog' | EN\: 'Open dialog' | PL: 'Otwórz dialog'
  686 = 'Operator' | EN\: 'Operator' | PL: 'Operator'
  148 = 'Option4' | EN\: 'Option4' | PL: 'Opcja4'
  232 = 'Option5' | EN\: 'Option5' | PL: 'Opcja5'
  756 = 'Option6' | EN\: 'Option6' | PL: 'Opcja6'
  426 = 'Ostatni czas cyklu' | EN\: 'Last cycle time' | PL: 'Ostatni czas cyklu'
  991 = 'p' | EN\: 'p' | PL: 'p'
  327 = 'P' | EN\: 'P' | PL: 'P'
  941 = 'POTWIERDŹ' | EN\: 'CONFIRM' | PL: 'POTWIERDŹ'
  1605 = 'Priorytet' | EN\: 'Priority' | PL: 'Priorytet'
  1631 = 'Przekroczony cykl' | EN\: 'Cycle exceeded' | PL: 'Przekroczony cykl'
  975 = 'q' | EN\: 'q' | PL: 'q'
  976 = 'Q' | EN\: 'Q' | PL: 'Q'
  981 = 'r' | EN\: 'r' | PL: 'r'
  982 = 'R' | EN\: 'R' | PL: 'R'
  106 = 'RESET' | EN\: 'RESET' | PL: 'RESET'
  296 = 'Reset' | EN\: 'Reset' | PL: 'Reset'
  221 = 'S' | EN\: 'S' | PL: 'S'
  609 = 's' | EN\: 's' | PL: 's'
  418 = 'Shift' | EN\: 'Shift' | PL: 'Shift'
  1066 = 'Show' | EN\: 'Show' | PL: 'Pokaż'
  419 = 'Space' | EN\: 'Space' | PL: 'Space'
  674 = 'support@beckhoff.pl' | EN\: 'suppoer@beckhoff.pl' | PL: 'support@beckhoff.pl'
  307 = 'System info' | EN\: 'System info' | PL: 'System info'
  1047 = 'System Info' | EN\: 'System Info' | PL: 'System Info'
  983 = 't' | EN\: 't' | PL: 't'
  984 = 'T' | EN\: 'T' | PL: 'T'
  869 = 'Table' | EN\: 'Table' | PL: 'Tabela'
  1639 = 'TAK' | EN\: 'Yes' | PL: 'TAK'
  95 = 'Task Info' | EN\: 'Task Info' | PL: 'TAsk Info'
  1327 = 'Trends' | EN\: 'Trends' | PL: 'Trendy'
  220 = 'U' | EN\: 'U' | PL: 'U'
  987 = 'u' | EN\: 'u' | PL: 'u'
  1645 = 'ul. Ruczajowa 15' | EN\: 'ul. Ruczajowa 15' | PL: 'ul. Ruczajowa 15'
  968 = 'User Management' | EN\: 'User Management' | PL: 'Zarządzaj '
  1185 = 'Ustaw' | EN\: 'Set' | PL: 'Set '
  781 = 'v' | EN\: 'v' | PL: 'v'
  782 = 'V' | EN\: 'V' | PL: 'V'
  977 = 'w' | EN\: 'w' | PL: 'w'
  978 = 'W' | EN\: 'W' | PL: 'W'
  1060 = 'Warning'
  446 = 'Wartość: %d' | EN\: 'Value: %d' | PL: 'Wartość: %d'
  156 = 'Wiersz: %d' | EN\: 'Line: %d' | PL: 'Wiersz: %d'
  1473 = 'www.beckhoff.pl' | EN\: 'www.beckhoff.pl' | PL: 'www.beckhoff.pl'
  777 = 'x' | EN\: 'x' | PL: 'x'
  778 = 'X' | EN\: 'X' | PL: 'X'
  775 = 'y' | EN\: 'y' | PL: 'y'
  776 = 'Y' | EN\: 'Y' | PL: 'Y'
  985 = 'z' | EN\: 'z' | PL: 'z'
  986 = 'Z' | EN\: 'Z' | PL: 'Z'
  1638 = 'Załadowano plik zapasowy' | EN\: 'Bakup file loaded' | PL: 'Załadowano plik zapasowy'
  874 = 'Załadowano poprawnie' | EN\: 'Loaded correctly' | PL: 'Załadowano poprawnie'
  459 = '[' | EN\: '[' | PL: '['
  470 = '\\' | EN\: '\\' | PL: '\\'
  466 = ']' | EN\: ']' | PL: ']'
  337 = '^' | EN\: '^' | PL: '^'
  789 = '_' | EN\: '_' | PL: '_'
  455 = '{' | EN\: '{' | PL: '{'
  420 = '|' | EN\: '|' | PL: '|'
  462 = '}' | EN\: '}' | PL: '}'
  333 = '~' | EN\: '~' | PL: '~'
  595 = '´' | EN\: "'" | PL: '´'
  428 = 'Średni czas cyklu' | EN\: 'Average cycle time' | PL: 'Średni czas cyklu'
END_TEXTLIST

// ---- VISUs/Internal/Keypad.TcVIS
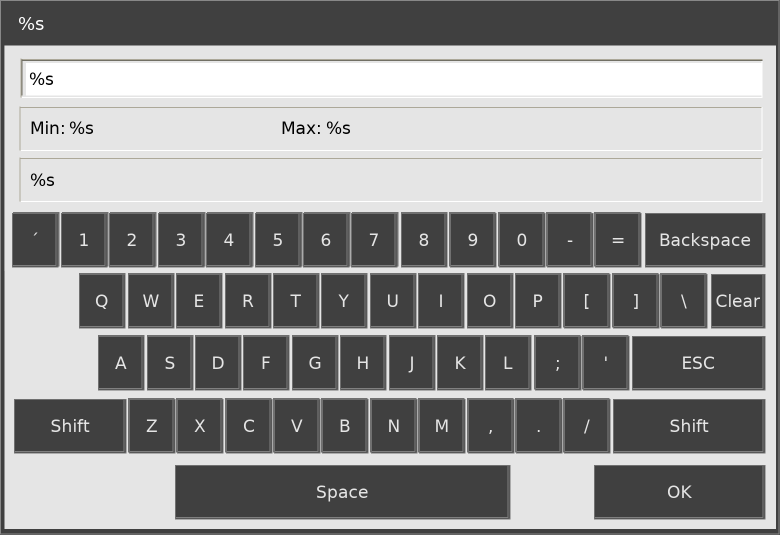
VISUALIZATION Keypad  // 780x535
VAR_INPUT
	stVariableValue 						: STRING;
	stMin 									: STRING;
	stMax 									: STRING;
	stTitle 								: STRING;
	flags 									: DWORD;
END_VAR
VAR
	bInit 									: BOOL;
	bShift 									: BOOL;
	stMessage 								: STRING;
	stOutputValue 							: STRING;
END_VAR
    Rectangle (5,201 772x70)
    Rectangle (3,271 775x62)
    Rectangle (3,333 775x63)
    Rectangle (3,396 775x62)
    Rectangle (3,455 775x75)
    Button (594,465 171x54), "OK"
        OnMouseDown: CloseDialog Dialog=Keypad, Result=OK, NumpadKeypad=True, NumpadKeypadSet=True
    Button (632,336 133x54), "ESC"
        OnMouseDown: CloseDialog Dialog=Keypad, Result=Cancel, NumpadKeypad=True, NumpadKeypadSet=True
    Button (711,274 54x54), "Clear"
        OnMouseDown: execute { stVariableValue := ''; stOutputValue := ''; }
    Button (645,213 120x54), "Backspace"
        OnMouseDown: execute { VisuDlg_CheckedBack(stOutputValue, stVariableValue, bInit); }
    Button (613,399 152x54), "Shift"
        OnMouseDown: toggle bShift
    Button (175,465 335x54), "Space"
        OnMouseDown: execute { VisuDlg_CheckedAppend(stOutputValue, stVariableValue, bInit, (flags AND VisuElems.Visu_InputFlags.Password) = 1, ' '); }
    Button (660,273 46x54), "|", invisible if: NOT bShift
        OnMouseDown: execute { VisuDlg_CheckedAppend(stOutputValue, stVariableValue, bInit, (flags AND VisuElems.Visu_InputFlags.Password) = 1, '|'); }
    Button (467,398 46x54), "<", invisible if: NOT bShift
        OnMouseDown: execute { VisuDlg_CheckedAppend(stOutputValue, stVariableValue, bInit, (flags AND VisuElems.Visu_InputFlags.Password) = 1, '<'); }
    Button (515,398 46x54), ">", invisible if: NOT bShift
        OnMouseDown: execute { VisuDlg_CheckedAppend(stOutputValue, stVariableValue, bInit, (flags AND VisuElems.Visu_InputFlags.Password) = 1, '>'); }
    Button (321,273 46x54), "y", invisible if: NOT bShift
        OnMouseDown: execute { VisuDlg_CheckedAppend(stOutputValue, stVariableValue, bInit, (flags AND VisuElems.Visu_InputFlags.Password) = 1, 'y'); }
    Button (321,274 46x54), "Y", invisible if: bShift
        OnMouseDown: execute { VisuDlg_CheckedAppend(stOutputValue, stVariableValue, bInit, (flags AND VisuElems.Visu_InputFlags.Password) = 1, 'Y'); }
    Button (176,398 46x54), "x", invisible if: NOT bShift
        OnMouseDown: execute { VisuDlg_CheckedAppend(stOutputValue, stVariableValue, bInit, (flags AND VisuElems.Visu_InputFlags.Password) = 1, 'x'); }
    Button (177,399 46x54), "X", invisible if: bShift
        OnMouseDown: execute { VisuDlg_CheckedAppend(stOutputValue, stVariableValue, bInit, (flags AND VisuElems.Visu_InputFlags.Password) = 1, 'X'); }
    Button (225,398 46x54), "c", invisible if: NOT bShift
        OnMouseDown: execute { VisuDlg_CheckedAppend(stOutputValue, stVariableValue, bInit, (flags AND VisuElems.Visu_InputFlags.Password) = 1, 'c'); }
    Button (226,399 46x54), "C", invisible if: bShift
        OnMouseDown: execute { VisuDlg_CheckedAppend(stOutputValue, stVariableValue, bInit, (flags AND VisuElems.Visu_InputFlags.Password) = 1, 'C'); }
    Button (273,398 46x54), "v", invisible if: NOT bShift
        OnMouseDown: execute { VisuDlg_CheckedAppend(stOutputValue, stVariableValue, bInit, (flags AND VisuElems.Visu_InputFlags.Password) = 1, 'v'); }
    Button (274,399 46x54), "V", invisible if: bShift
        OnMouseDown: execute { VisuDlg_CheckedAppend(stOutputValue, stVariableValue, bInit, (flags AND VisuElems.Visu_InputFlags.Password) = 1, 'V'); }
    Button (321,398 46x54), "b", invisible if: NOT bShift
        OnMouseDown: execute { VisuDlg_CheckedAppend(stOutputValue, stVariableValue, bInit, (flags AND VisuElems.Visu_InputFlags.Password) = 1, 'b'); }
    Button (322,399 46x54), "B", invisible if: bShift
        OnMouseDown: execute { VisuDlg_CheckedAppend(stOutputValue, stVariableValue, bInit, (flags AND VisuElems.Visu_InputFlags.Password) = 1, 'B'); }
    Button (370,398 46x54), "n", invisible if: NOT bShift
        OnMouseDown: execute { VisuDlg_CheckedAppend(stOutputValue, stVariableValue, bInit, (flags AND VisuElems.Visu_InputFlags.Password) = 1, 'n'); }
    Button (371,399 46x54), "N", invisible if: bShift
        OnMouseDown: execute { VisuDlg_CheckedAppend(stOutputValue, stVariableValue, bInit, (flags AND VisuElems.Visu_InputFlags.Password) = 1, 'N'); }
    Button (418,398 46x54), "m", invisible if: NOT bShift
        OnMouseDown: execute { VisuDlg_CheckedAppend(stOutputValue, stVariableValue, bInit, (flags AND VisuElems.Visu_InputFlags.Password) = 1, 'm'); }
    Button (419,399 46x54), "M", invisible if: bShift
        OnMouseDown: execute { VisuDlg_CheckedAppend(stOutputValue, stVariableValue, bInit, (flags AND VisuElems.Visu_InputFlags.Password) = 1, 'M'); }
    Button (534,335 46x54), ":", invisible if: NOT bShift
        OnMouseDown: execute { VisuDlg_CheckedAppend(stOutputValue, stVariableValue, bInit, (flags AND VisuElems.Visu_InputFlags.Password) = 1, ':'); }
    Button (546,212 45x54), "_", invisible if: NOT bShift
        OnMouseDown: execute { VisuDlg_CheckedAppend(stOutputValue, stVariableValue, bInit, (flags AND VisuElems.Visu_InputFlags.Password) = 1, '_'); }
    Button (98,335 46x54), "a", invisible if: NOT bShift
        OnMouseDown: execute { VisuDlg_CheckedAppend(stOutputValue, stVariableValue, bInit, (flags AND VisuElems.Visu_InputFlags.Password) = 1, 'a'); }
    Button (98,336 46x54), "A", invisible if: bShift
        OnMouseDown: execute { VisuDlg_CheckedAppend(stOutputValue, stVariableValue, bInit, (flags AND VisuElems.Visu_InputFlags.Password) = 1, 'A'); }
    Button (147,335 46x54), "s", invisible if: NOT bShift
        OnMouseDown: execute { VisuDlg_CheckedAppend(stOutputValue, stVariableValue, bInit, (flags AND VisuElems.Visu_InputFlags.Password) = 1, 's'); }
    Button (147,336 46x54), "S", invisible if: bShift
        OnMouseDown: execute { VisuDlg_CheckedAppend(stOutputValue, stVariableValue, bInit, (flags AND VisuElems.Visu_InputFlags.Password) = 1, 'S'); }
    Button (195,335 46x54), "d", invisible if: NOT bShift
        OnMouseDown: execute { VisuDlg_CheckedAppend(stOutputValue, stVariableValue, bInit, (flags AND VisuElems.Visu_InputFlags.Password) = 1, 'd'); }
    Button (195,336 46x54), "D", invisible if: bShift
        OnMouseDown: execute { VisuDlg_CheckedAppend(stOutputValue, stVariableValue, bInit, (flags AND VisuElems.Visu_InputFlags.Password) = 1, 'D'); }
    Button (243,335 46x54), "f", invisible if: NOT bShift
        OnMouseDown: execute { VisuDlg_CheckedAppend(stOutputValue, stVariableValue, bInit, (flags AND VisuElems.Visu_InputFlags.Password) = 1, 'f'); }
    Button (243,336 46x54), "F", invisible if: bShift
        OnMouseDown: execute { VisuDlg_CheckedAppend(stOutputValue, stVariableValue, bInit, (flags AND VisuElems.Visu_InputFlags.Password) = 1, 'F'); }
    Button (292,335 46x54), "g", invisible if: NOT bShift
        OnMouseDown: execute { VisuDlg_CheckedAppend(stOutputValue, stVariableValue, bInit, (flags AND VisuElems.Visu_InputFlags.Password) = 1, 'g'); }
    Button (292,336 46x54), "G", invisible if: bShift
        OnMouseDown: execute { VisuDlg_CheckedAppend(stOutputValue, stVariableValue, bInit, (flags AND VisuElems.Visu_InputFlags.Password) = 1, 'G'); }
    Button (340,335 46x54), "h", invisible if: NOT bShift
        OnMouseDown: execute { VisuDlg_CheckedAppend(stOutputValue, stVariableValue, bInit, (flags AND VisuElems.Visu_InputFlags.Password) = 1, 'h'); }
    Button (340,336 46x54), "H", invisible if: bShift
        OnMouseDown: execute { VisuDlg_CheckedAppend(stOutputValue, stVariableValue, bInit, (flags AND VisuElems.Visu_InputFlags.Password) = 1, 'H'); }
    Button (389,335 46x54), "j", invisible if: NOT bShift
        OnMouseDown: execute { VisuDlg_CheckedAppend(stOutputValue, stVariableValue, bInit, (flags AND VisuElems.Visu_InputFlags.Password) = 1, 'j'); }
    Button (389,336 46x54), "J", invisible if: bShift
        OnMouseDown: execute { VisuDlg_CheckedAppend(stOutputValue, stVariableValue, bInit, (flags AND VisuElems.Visu_InputFlags.Password) = 1, 'J'); }
    Button (437,335 46x54), "k", invisible if: NOT bShift
        OnMouseDown: execute { VisuDlg_CheckedAppend(stOutputValue, stVariableValue, bInit, (flags AND VisuElems.Visu_InputFlags.Password) = 1, 'k'); }
    Button (437,336 46x54), "K", invisible if: bShift
        OnMouseDown: execute { VisuDlg_CheckedAppend(stOutputValue, stVariableValue, bInit, (flags AND VisuElems.Visu_InputFlags.Password) = 1, 'K'); }
    Button (485,335 46x54), "l", invisible if: NOT bShift
        OnMouseDown: execute { VisuDlg_CheckedAppend(stOutputValue, stVariableValue, bInit, (flags AND VisuElems.Visu_InputFlags.Password) = 1, 'l'); }
    Button (485,336 46x54), "L", invisible if: bShift
        OnMouseDown: execute { VisuDlg_CheckedAppend(stOutputValue, stVariableValue, bInit, (flags AND VisuElems.Visu_InputFlags.Password) = 1, 'L'); }
    Button (159,212 46x54), "#", invisible if: NOT bShift
        OnMouseDown: execute { VisuDlg_CheckedAppend(stOutputValue, stVariableValue, bInit, (flags AND VisuElems.Visu_InputFlags.Password) = 1, '#'); }
    Button (110,212 46x54), "@", invisible if: NOT bShift
        OnMouseDown: execute { VisuDlg_CheckedAppend(stOutputValue, stVariableValue, bInit, (flags AND VisuElems.Visu_InputFlags.Password) = 1, '@'); }
    Button (79,273 46x54), "q", invisible if: NOT bShift
        OnMouseDown: execute { VisuDlg_CheckedAppend(stOutputValue, stVariableValue, bInit, (flags AND VisuElems.Visu_InputFlags.Password) = 1, 'q'); }
    Button (79,274 46x54), "Q", invisible if: bShift
        OnMouseDown: execute { VisuDlg_CheckedAppend(stOutputValue, stVariableValue, bInit, (flags AND VisuElems.Visu_InputFlags.Password) = 1, 'Q'); }
    Button (128,273 46x54), "w", invisible if: NOT bShift
        OnMouseDown: execute { VisuDlg_CheckedAppend(stOutputValue, stVariableValue, bInit, (flags AND VisuElems.Visu_InputFlags.Password) = 1, 'w'); }
    Button (128,274 46x54), "W", invisible if: bShift
        OnMouseDown: execute { VisuDlg_CheckedAppend(stOutputValue, stVariableValue, bInit, (flags AND VisuElems.Visu_InputFlags.Password) = 1, 'W'); }
    Button (176,273 46x54), "e", invisible if: NOT bShift
        OnMouseDown: execute { VisuDlg_CheckedAppend(stOutputValue, stVariableValue, bInit, (flags AND VisuElems.Visu_InputFlags.Password) = 1, 'e'); }
    Button (176,274 46x54), "E", invisible if: bShift
        OnMouseDown: execute { VisuDlg_CheckedAppend(stOutputValue, stVariableValue, bInit, (flags AND VisuElems.Visu_InputFlags.Password) = 1, 'E'); }
    Button (225,273 46x54), "r", invisible if: NOT bShift
        OnMouseDown: execute { VisuDlg_CheckedAppend(stOutputValue, stVariableValue, bInit, (flags AND VisuElems.Visu_InputFlags.Password) = 1, 'r'); }
    Button (225,274 46x54), "R", invisible if: bShift
        OnMouseDown: execute { VisuDlg_CheckedAppend(stOutputValue, stVariableValue, bInit, (flags AND VisuElems.Visu_InputFlags.Password) = 1, 'R'); }
    Button (273,273 46x54), "t", invisible if: NOT bShift
        OnMouseDown: execute { VisuDlg_CheckedAppend(stOutputValue, stVariableValue, bInit, (flags AND VisuElems.Visu_InputFlags.Password) = 1, 't'); }
    Button (273,274 46x54), "T", invisible if: bShift
        OnMouseDown: execute { VisuDlg_CheckedAppend(stOutputValue, stVariableValue, bInit, (flags AND VisuElems.Visu_InputFlags.Password) = 1, 'T'); }
    Button (128,398 46x54), "z", invisible if: NOT bShift
        OnMouseDown: execute { VisuDlg_CheckedAppend(stOutputValue, stVariableValue, bInit, (flags AND VisuElems.Visu_InputFlags.Password) = 1, 'z'); }
    Button (129,399 46x54), "Z", invisible if: bShift
        OnMouseDown: execute { VisuDlg_CheckedAppend(stOutputValue, stVariableValue, bInit, (flags AND VisuElems.Visu_InputFlags.Password) = 1, 'Z'); }
    Button (370,273 46x54), "u", invisible if: NOT bShift
        OnMouseDown: execute { VisuDlg_CheckedAppend(stOutputValue, stVariableValue, bInit, (flags AND VisuElems.Visu_InputFlags.Password) = 1, 'u'); }
    Button (370,274 46x54), "U", invisible if: bShift
        OnMouseDown: execute { VisuDlg_CheckedAppend(stOutputValue, stVariableValue, bInit, (flags AND VisuElems.Visu_InputFlags.Password) = 1, 'U'); }
    Button (418,273 46x54), "i", invisible if: NOT bShift
        OnMouseDown: execute { VisuDlg_CheckedAppend(stOutputValue, stVariableValue, bInit, (flags AND VisuElems.Visu_InputFlags.Password) = 1, 'i'); }
    Button (418,274 46x54), "I", invisible if: bShift
        OnMouseDown: execute { VisuDlg_CheckedAppend(stOutputValue, stVariableValue, bInit, (flags AND VisuElems.Visu_InputFlags.Password) = 1, 'I'); }
    Button (467,273 46x54), "o", invisible if: NOT bShift
        OnMouseDown: execute { VisuDlg_CheckedAppend(stOutputValue, stVariableValue, bInit, (flags AND VisuElems.Visu_InputFlags.Password) = 1, 'o'); }
    Button (467,274 46x54), "O", invisible if: bShift
        OnMouseDown: execute { VisuDlg_CheckedAppend(stOutputValue, stVariableValue, bInit, (flags AND VisuElems.Visu_InputFlags.Password) = 1, 'O'); }
    Button (515,273 46x54), "p", invisible if: NOT bShift
        OnMouseDown: execute { VisuDlg_CheckedAppend(stOutputValue, stVariableValue, bInit, (flags AND VisuElems.Visu_InputFlags.Password) = 1, 'p'); }
    Button (515,274 46x54), "P", invisible if: bShift
        OnMouseDown: execute { VisuDlg_CheckedAppend(stOutputValue, stVariableValue, bInit, (flags AND VisuElems.Visu_InputFlags.Password) = 1, 'P'); }
    Button (594,212 46x54), "+", invisible if: NOT bShift
        OnMouseDown: execute { VisuDlg_CheckedAppend(stOutputValue, stVariableValue, bInit, (flags AND VisuElems.Visu_InputFlags.Password) = 1, '+'); }
    Button (401,212 46x54), "*", invisible if: NOT bShift
        OnMouseDown: execute { VisuDlg_CheckedAppend(stOutputValue, stVariableValue, bInit, (flags AND VisuElems.Visu_InputFlags.Password) = 1, '*'); }
    Button (13,212 46x54), "~", invisible if: NOT bShift
        OnMouseDown: execute { VisuDlg_CheckedAppend(stOutputValue, stVariableValue, bInit, (flags AND VisuElems.Visu_InputFlags.Password) = 1, '~'); }
    Button (304,212 46x54), "^", invisible if: NOT bShift
        OnMouseDown: execute { VisuDlg_CheckedAppend(stOutputValue, stVariableValue, bInit, (flags AND VisuElems.Visu_InputFlags.Password) = 1, '^'); }
    Button (62,212 46x54), "!", invisible if: NOT bShift
        OnMouseDown: execute { VisuDlg_CheckedAppend(stOutputValue, stVariableValue, bInit, (flags AND VisuElems.Visu_InputFlags.Password) = 1, '!'); }
    Button (582,335 46x54), """, invisible if: NOT bShift
        OnMouseDown: execute { VisuDlg_CheckedAppend(stOutputValue, stVariableValue, bInit, (flags AND VisuElems.Visu_InputFlags.Password) = 1, '"'); }
    Button (207,212 46x54), "$", invisible if: NOT bShift
        OnMouseDown: execute { VisuDlg_CheckedAppend(stOutputValue, stVariableValue, bInit, (flags AND VisuElems.Visu_InputFlags.Password) = 1, '$$'); }
    Button (256,212 46x54), "%", invisible if: NOT bShift
        OnMouseDown: execute { VisuDlg_CheckedAppend(stOutputValue, stVariableValue, bInit, (flags AND VisuElems.Visu_InputFlags.Password) = 1, '%'); }
    Button (352,212 46x54), "&", invisible if: NOT bShift
        OnMouseDown: execute { VisuDlg_CheckedAppend(stOutputValue, stVariableValue, bInit, (flags AND VisuElems.Visu_InputFlags.Password) = 1, '&'); }
    Button (449,212 46x54), "(", invisible if: NOT bShift
        OnMouseDown: execute { VisuDlg_CheckedAppend(stOutputValue, stVariableValue, bInit, (flags AND VisuElems.Visu_InputFlags.Password) = 1, '('); }
    Button (498,212 46x54), ")", invisible if: NOT bShift
        OnMouseDown: execute { VisuDlg_CheckedAppend(stOutputValue, stVariableValue, bInit, (flags AND VisuElems.Visu_InputFlags.Password) = 1, ')'); }
    Button (563,398 46x54), "?", invisible if: NOT bShift
        OnMouseDown: execute { VisuDlg_CheckedAppend(stOutputValue, stVariableValue, bInit, (flags AND VisuElems.Visu_InputFlags.Password) = 1, '?'); }
    Rectangle (5,104 773x97)
    Rectangle (27,164 734x32), "%s", text variable: stMessage
    Rectangle (5,42 773x62)
    Rectangle (776,0 4x530)
    Rectangle (0,2 4x527)
    Rectangle (0,529 780x6)
    Polyline (20,201) (20,158) (762,158)
    Polyline (20,150) (20,107) (762,107)
    Polyline (21,97) (21,59) (762,59)
    Polyline (21,201) (762,201) (762,158)
    Polyline (21,150) (762,150) (762,107)
    Polyline (22,97) (762,97) (762,60)
    Rectangle (0,0 779x45)
    Rectangle (15,8 757x32), "%s", text variable: stTitle
    Polyline (22,95) (22,60) (762,60)
    Rectangle (26,63 736x32), "%s", text variable: stOutputValue
    Rectangle (27,112 42x32), "Min:", text variable: stMin, invisible if: LEN(stMin) = 0
    Rectangle (66,112 157x32), "%s", text variable: stMin, invisible if: LEN(stMin) = 0
    Rectangle (278,112 45x32), "Max:", text variable: stMin, invisible if: LEN(stMax) = 0
    Rectangle (323,112 217x32), "%s", text variable: stMax, invisible if: LEN(stMax) = 0
    Button (12,213 46x54), "´", invisible if: bShift
        OnMouseDown: execute { VisuDlg_CheckedAppend(stOutputValue, stVariableValue, bInit, (flags AND VisuElems.Visu_InputFlags.Password) = 1, '´'); }
    Button (61,213 46x54), "1", invisible if: bShift
        OnMouseDown: execute { VisuDlg_CheckedAppend(stOutputValue, stVariableValue, bInit, (flags AND VisuElems.Visu_InputFlags.Password) = 1, '1'); }
    Button (109,213 46x54), "2", invisible if: bShift
        OnMouseDown: execute { VisuDlg_CheckedAppend(stOutputValue, stVariableValue, bInit, (flags AND VisuElems.Visu_InputFlags.Password) = 1, '2'); }
    Button (158,213 46x54), "3", invisible if: bShift
        OnMouseDown: execute { VisuDlg_CheckedAppend(stOutputValue, stVariableValue, bInit, (flags AND VisuElems.Visu_InputFlags.Password) = 1, '3'); }
    Button (206,213 46x54), "4", invisible if: bShift
        OnMouseDown: execute { VisuDlg_CheckedAppend(stOutputValue, stVariableValue, bInit, (flags AND VisuElems.Visu_InputFlags.Password) = 1, '4'); }
    Button (255,213 46x54), "5", invisible if: bShift
        OnMouseDown: execute { VisuDlg_CheckedAppend(stOutputValue, stVariableValue, bInit, (flags AND VisuElems.Visu_InputFlags.Password) = 1, '5'); }
    Button (303,213 46x54), "6", invisible if: bShift
        OnMouseDown: execute { VisuDlg_CheckedAppend(stOutputValue, stVariableValue, bInit, (flags AND VisuElems.Visu_InputFlags.Password) = 1, '6'); }
    Button (351,213 46x54), "7", invisible if: bShift
        OnMouseDown: execute { VisuDlg_CheckedAppend(stOutputValue, stVariableValue, bInit, (flags AND VisuElems.Visu_InputFlags.Password) = 1, '7'); }
    Button (401,213 46x54), "8", invisible if: bShift
        OnMouseDown: execute { VisuDlg_CheckedAppend(stOutputValue, stVariableValue, bInit, (flags AND VisuElems.Visu_InputFlags.Password) = 1, '8'); }
    Button (450,213 46x54), "9", invisible if: bShift
        OnMouseDown: execute { VisuDlg_CheckedAppend(stOutputValue, stVariableValue, bInit, (flags AND VisuElems.Visu_InputFlags.Password) = 1, '9'); }
    Button (499,213 46x54), "0", invisible if: bShift
        OnMouseDown: execute { VisuDlg_CheckedAppend(stOutputValue, stVariableValue, bInit, (flags AND VisuElems.Visu_InputFlags.Password) = 1, '0'); }
    Button (547,213 46x54), "-", invisible if: bShift
        OnMouseDown: execute { VisuDlg_CheckedAppend(stOutputValue, stVariableValue, bInit, (flags AND VisuElems.Visu_InputFlags.Password) = 1, '-'); }
    Button (595,213 46x54), "=", invisible if: bShift
        OnMouseDown: execute { VisuDlg_CheckedAppend(stOutputValue, stVariableValue, bInit, (flags AND VisuElems.Visu_InputFlags.Password) = 1, '='); }
    Button (563,273 46x54), "{", invisible if: NOT bShift
        OnMouseDown: execute { VisuDlg_CheckedAppend(stOutputValue, stVariableValue, bInit, (flags AND VisuElems.Visu_InputFlags.Password) = 1, '{'); }
    Button (564,274 46x54), "[", invisible if: bShift
        OnMouseDown: execute { VisuDlg_CheckedAppend(stOutputValue, stVariableValue, bInit, (flags AND VisuElems.Visu_InputFlags.Password) = 1, '['); }
    Button (612,273 46x54), "}", invisible if: NOT bShift
        OnMouseDown: execute { VisuDlg_CheckedAppend(stOutputValue, stVariableValue, bInit, (flags AND VisuElems.Visu_InputFlags.Password) = 1, '}'); }
    Button (613,274 46x54), "]", invisible if: bShift
        OnMouseDown: execute { VisuDlg_CheckedAppend(stOutputValue, stVariableValue, bInit, (flags AND VisuElems.Visu_InputFlags.Password) = 1, ']'); }
    Button (661,274 46x54), "\", invisible if: bShift
        OnMouseDown: execute { VisuDlg_CheckedAppend(stOutputValue, stVariableValue, bInit, (flags AND VisuElems.Visu_InputFlags.Password) = 1, '\'); }
    Button (535,336 46x54), ";", invisible if: bShift
        OnMouseDown: execute { VisuDlg_CheckedAppend(stOutputValue, stVariableValue, bInit, (flags AND VisuElems.Visu_InputFlags.Password) = 1, ';'); }
    Button (583,336 46x54), "'", invisible if: bShift
        OnMouseDown: execute { VisuDlg_CheckedAppend(stOutputValue, stVariableValue, bInit, (flags AND VisuElems.Visu_InputFlags.Password) = 1, '$''); }
    Button (468,399 46x54), ",", invisible if: bShift
        OnMouseDown: execute { VisuDlg_CheckedAppend(stOutputValue, stVariableValue, bInit, (flags AND VisuElems.Visu_InputFlags.Password) = 1, ','); }
    Button (516,399 46x54), ".", invisible if: bShift
        OnMouseDown: execute { VisuDlg_CheckedAppend(stOutputValue, stVariableValue, bInit, (flags AND VisuElems.Visu_InputFlags.Password) = 1, '.'); }
    Button (564,399 46x54), "/", invisible if: bShift
        OnMouseDown: execute { VisuDlg_CheckedAppend(stOutputValue, stVariableValue, bInit, (flags AND VisuElems.Visu_InputFlags.Password) = 1, '/'); }
    Button (14,399 112x54), "Shift"
        OnMouseDown: toggle bShift
    hotkey HotkeyInput Id=481083523072, Key=KeyDown=True, KeyName=BACKSPACE, ActionToExecute=Action=STSnippet=VisuDlg_CheckedBack(stOutputValue, stVariableValue, bInit);, VisuElemId=-1
    hotkey HotkeyInput Id=481084571648, Key=KeyDown=True, KeyName=DELETE, ActionToExecute=Action=STSnippet=stVariableValue := ''; stOutputValue := '';, VisuElemId=-1
    hotkey HotkeyInput Id=481085620224, Key=KeyDown=True, KeyName=ESCAPE, ActionToExecute=Action=Dialog=Keypad, Result=Cancel, NumpadKeypad=True, NumpadKeypadSet=True, VisuElemId=-1
    hotkey HotkeyInput Id=481086668800, Key=KeyDown=True, KeyName=SPACE, ActionToExecute=Action=STSnippet=VisuDlg_CheckedAppend(stOutputValue, stVariableValue, bInit, (flags AND VisuElems.Visu_InputFlags.Password) = 1, ' ');, VisuElemId=-1
    hotkey HotkeyInput Id=481087717376, Key=Modifiers=1, KeyDown=True, KeyName=SPACE, ActionToExecute=Action=ToggleVariable=bShift, VisuElemId=-1
    hotkey HotkeyInput Id=481088765952, Key=KeyDown=True, KeyName=RETURN_KEY, ActionToExecute=Action=Dialog=Keypad, Result=OK, NumpadKeypad=True, NumpadKeypadSet=True, VisuElemId=-1
    hotkey HotkeyInput Id=481089814528, Key=KeyDown=True, KeyName=1, ActionToExecute=Action=STSnippet=IF bShift THEN VisuDlg_CheckedAppend(stOutputValue, stVariableValue, bInit, (flags AND VisuElems.Visu_InputFlags.Password) = 1, '!'); ELSE VisuDlg_CheckedAppend(stOutputValue, stVariableValue, bInit, (flags AND VisuElems.Visu_InputFlags.Password) = 1, '1'); END_IF, VisuElemId=-1
    hotkey HotkeyInput Id=481090863104, Key=KeyDown=True, KeyName=2, ActionToExecute=Action=STSnippet=IF bShift THEN VisuDlg_CheckedAppend(stOutputValue, stVariableValue, bInit, (flags AND VisuElems.Visu_InputFlags.Password) = 1, '@'); ELSE VisuDlg_CheckedAppend(stOutputValue, stVariableValue, bInit, (flags AND VisuElems.Visu_InputFlags.Password) = 1, '2'); END_IF, VisuElemId=-1
    hotkey HotkeyInput Id=481091911680, Key=KeyDown=True, KeyName=3, ActionToExecute=Action=STSnippet=IF bShift THEN VisuDlg_CheckedAppend(stOutputValue, stVariableValue, bInit, (flags AND VisuElems.Visu_InputFlags.Password) = 1, '#'); ELSE VisuDlg_CheckedAppend(stOutputValue, stVariableValue, bInit, (flags AND VisuElems.Visu_InputFlags.Password) = 1, '3'); END_IF, VisuElemId=-1
    hotkey HotkeyInput Id=481092960256, Key=KeyDown=True, KeyName=4, ActionToExecute=Action=STSnippet=IF bShift THEN VisuDlg_CheckedAppend(stOutputValue, stVariableValue, bInit, (flags AND VisuElems.Visu_InputFlags.Password) = 1, '$$'); ELSE VisuDlg_CheckedAppend(stOutputValue, stVariableValue, bInit, (flags AND VisuElems.Visu_InputFlags.Password) = 1, '4'); END_IF, VisuElemId=-1
    hotkey HotkeyInput Id=481094008832, Key=KeyDown=True, KeyName=5, ActionToExecute=Action=STSnippet=IF bShift THEN VisuDlg_CheckedAppend(stOutputValue, stVariableValue, bInit, (flags AND VisuElems.Visu_InputFlags.Password) = 1, '%'); ELSE VisuDlg_CheckedAppend(stOutputValue, stVariableValue, bInit, (flags AND VisuElems.Visu_InputFlags.Password) = 1, '5'); END_IF, VisuElemId=-1
    hotkey HotkeyInput Id=481095057408, Key=KeyDown=True, KeyName=6, ActionToExecute=Action=STSnippet=IF bShift THEN VisuDlg_CheckedAppend(stOutputValue, stVariableValue, bInit, (flags AND VisuElems.Visu_InputFlags.Password) = 1, '^'); ELSE VisuDlg_CheckedAppend(stOutputValue, stVariableValue, bInit, (flags AND VisuElems.Visu_InputFlags.Password) = 1, '6'); END_IF, VisuElemId=-1
    hotkey HotkeyInput Id=481096105984, Key=KeyDown=True, KeyName=7, ActionToExecute=Action=STSnippet=IF bShift THEN VisuDlg_CheckedAppend(stOutputValue, stVariableValue, bInit, (flags AND VisuElems.Visu_InputFlags.Password) = 1, '&'); ELSE VisuDlg_CheckedAppend(stOutputValue, stVariableValue, bInit, (flags AND VisuElems.Visu_InputFlags.Password) = 1, '7'); END_IF, VisuElemId=-1
    hotkey HotkeyInput Id=481097154560, Key=KeyDown=True, KeyName=8, ActionToExecute=Action=STSnippet=IF bShift THEN VisuDlg_CheckedAppend(stOutputValue, stVariableValue, bInit, (flags AND VisuElems.Visu_InputFlags.Password) = 1, '*'); ELSE VisuDlg_CheckedAppend(stOutputValue, stVariableValue, bInit, (flags AND VisuElems.Visu_InputFlags.Password) = 1, '8'); END_IF, VisuElemId=-1
    hotkey HotkeyInput Id=481098203136, Key=KeyDown=True, KeyName=9, ActionToExecute=Action=STSnippet=IF bShift THEN VisuDlg_CheckedAppend(stOutputValue, stVariableValue, bInit, (flags AND VisuElems.Visu_InputFlags.Password) = 1, '('); ELSE VisuDlg_CheckedAppend(stOutputValue, stVariableValue, bInit, (flags AND VisuElems.Visu_InputFlags.Password) = 1, '9'); END_IF, VisuElemId=-1
    hotkey HotkeyInput Id=481099251712, Key=KeyDown=True, KeyName=0, ActionToExecute=Action=STSnippet=IF bShift THEN VisuDlg_CheckedAppend(stOutputValue, stVariableValue, bInit, (flags AND VisuElems.Visu_InputFlags.Password) = 1, ')'); ELSE VisuDlg_CheckedAppend(stOutputValue, stVariableValue, bInit, (flags AND VisuElems.Visu_InputFlags.Password) = 1, '0'); END_IF, VisuElemId=-1
    hotkey HotkeyInput Id=481100300288, Key=KeyDown=True, KeyName=SUBTRACT, ActionToExecute=Action=STSnippet=IF bShift THEN VisuDlg_CheckedAppend(stOutputValue, stVariableValue, bInit, (flags AND VisuElems.Visu_InputFlags.Password) = 1, '_'); ELSE VisuDlg_CheckedAppend(stOutputValue, stVariableValue, bInit, (flags AND VisuElems.Visu_InputFlags.Password) = 1, '-'); END_IF, VisuElemId=-1
    hotkey HotkeyInput Id=481101348864, Key=KeyDown=True, KeyName=ADDITION, ActionToExecute=Action=STSnippet=IF bShift THEN VisuDlg_CheckedAppend(stOutputValue, stVariableValue, bInit, (flags AND VisuElems.Visu_InputFlags.Password) = 1, '='); ELSE VisuDlg_CheckedAppend(stOutputValue, stVariableValue, bInit, (flags AND VisuElems.Visu_InputFlags.Password) = 1, '+'); END_IF, VisuElemId=-1
    hotkey HotkeyInput Id=481102397440, Key=KeyDown=True, KeyName=Q, ActionToExecute=Action=STSnippet=IF bShift THEN VisuDlg_CheckedAppend(stOutputValue, stVariableValue, bInit, (flags AND VisuElems.Visu_InputFlags.Password) = 1, 'q'); ELSE VisuDlg_CheckedAppend(stOutputValue, stVariableValue, bInit, (flags AND VisuElems.Visu_InputFlags.Password) = 1, 'Q'); END_IF, VisuElemId=-1
    hotkey HotkeyInput Id=481103446016, Key=KeyDown=True, KeyName=W, ActionToExecute=Action=STSnippet=IF bShift THEN VisuDlg_CheckedAppend(stOutputValue, stVariableValue, bInit, (flags AND VisuElems.Visu_InputFlags.Password) = 1, 'w'); ELSE VisuDlg_CheckedAppend(stOutputValue, stVariableValue, bInit, (flags AND VisuElems.Visu_InputFlags.Password) = 1, 'W'); END_IF, VisuElemId=-1
    hotkey HotkeyInput Id=481104494592, Key=KeyDown=True, KeyName=E, ActionToExecute=Action=STSnippet=IF bShift THEN VisuDlg_CheckedAppend(stOutputValue, stVariableValue, bInit, (flags AND VisuElems.Visu_InputFlags.Password) = 1, 'e'); ELSE VisuDlg_CheckedAppend(stOutputValue, stVariableValue, bInit, (flags AND VisuElems.Visu_InputFlags.Password) = 1, 'E'); END_IF, VisuElemId=-1
    hotkey HotkeyInput Id=481105543168, Key=KeyDown=True, KeyName=R, ActionToExecute=Action=STSnippet=IF bShift THEN VisuDlg_CheckedAppend(stOutputValue, stVariableValue, bInit, (flags AND VisuElems.Visu_InputFlags.Password) = 1, 'r'); ELSE VisuDlg_CheckedAppend(stOutputValue, stVariableValue, bInit, (flags AND VisuElems.Visu_InputFlags.Password) = 1, 'R'); END_IF, VisuElemId=-1
    hotkey HotkeyInput Id=481106591744, Key=KeyDown=True, KeyName=T, ActionToExecute=Action=STSnippet=IF bShift THEN VisuDlg_CheckedAppend(stOutputValue, stVariableValue, bInit, (flags AND VisuElems.Visu_InputFlags.Password) = 1, 't'); ELSE VisuDlg_CheckedAppend(stOutputValue, stVariableValue, bInit, (flags AND VisuElems.Visu_InputFlags.Password) = 1, 'T'); END_IF, VisuElemId=-1
    hotkey HotkeyInput Id=481107640320, Key=KeyDown=True, KeyName=Y, ActionToExecute=Action=STSnippet=IF bShift THEN VisuDlg_CheckedAppend(stOutputValue, stVariableValue, bInit, (flags AND VisuElems.Visu_InputFlags.Password) = 1, 'y'); ELSE VisuDlg_CheckedAppend(stOutputValue, stVariableValue, bInit, (flags AND VisuElems.Visu_InputFlags.Password) = 1, 'Y'); END_IF, VisuElemId=-1
    hotkey HotkeyInput Id=481108688896, Key=KeyDown=True, KeyName=U, ActionToExecute=Action=STSnippet=IF bShift THEN VisuDlg_CheckedAppend(stOutputValue, stVariableValue, bInit, (flags AND VisuElems.Visu_InputFlags.Password) = 1, 'u'); ELSE VisuDlg_CheckedAppend(stOutputValue, stVariableValue, bInit, (flags AND VisuElems.Visu_InputFlags.Password) = 1, 'U'); END_IF, VisuElemId=-1
    hotkey HotkeyInput Id=481109737472, Key=KeyDown=True, KeyName=I, ActionToExecute=Action=STSnippet=IF bShift THEN VisuDlg_CheckedAppend(stOutputValue, stVariableValue, bInit, (flags AND VisuElems.Visu_InputFlags.Password) = 1, 'i'); ELSE VisuDlg_CheckedAppend(stOutputValue, stVariableValue, bInit, (flags AND VisuElems.Visu_InputFlags.Password) = 1, 'I'); END_IF, VisuElemId=-1
    hotkey HotkeyInput Id=481110786048, Key=KeyDown=True, KeyName=O, ActionToExecute=Action=STSnippet=IF bShift THEN VisuDlg_CheckedAppend(stOutputValue, stVariableValue, bInit, (flags AND VisuElems.Visu_InputFlags.Password) = 1, 'o'); ELSE VisuDlg_CheckedAppend(stOutputValue, stVariableValue, bInit, (flags AND VisuElems.Visu_InputFlags.Password) = 1, 'O'); END_IF, VisuElemId=-1
    hotkey HotkeyInput Id=481111834624, Key=KeyDown=True, KeyName=P, ActionToExecute=Action=STSnippet=IF bShift THEN VisuDlg_CheckedAppend(stOutputValue, stVariableValue, bInit, (flags AND VisuElems.Visu_InputFlags.Password) = 1, 'p'); ELSE VisuDlg_CheckedAppend(stOutputValue, stVariableValue, bInit, (flags AND VisuElems.Visu_InputFlags.Password) = 1, 'P'); END_IF, VisuElemId=-1
    hotkey HotkeyInput Id=481112883200, Key=KeyDown=True, KeyName=A, ActionToExecute=Action=STSnippet=IF bShift THEN VisuDlg_CheckedAppend(stOutputValue, stVariableValue, bInit, (flags AND VisuElems.Visu_InputFlags.Password) = 1, 'a'); ELSE VisuDlg_CheckedAppend(stOutputValue, stVariableValue, bInit, (flags AND VisuElems.Visu_InputFlags.Password) = 1, 'A'); END_IF, VisuElemId=-1
    hotkey HotkeyInput Id=481113931776, Key=KeyDown=True, KeyName=S, ActionToExecute=Action=STSnippet=IF bShift THEN VisuDlg_CheckedAppend(stOutputValue, stVariableValue, bInit, (flags AND VisuElems.Visu_InputFlags.Password) = 1, 's'); ELSE VisuDlg_CheckedAppend(stOutputValue, stVariableValue, bInit, (flags AND VisuElems.Visu_InputFlags.Password) = 1, 'S'); END_IF, VisuElemId=-1
    hotkey HotkeyInput Id=481114980352, Key=KeyDown=True, KeyName=D, ActionToExecute=Action=STSnippet=IF bShift THEN VisuDlg_CheckedAppend(stOutputValue, stVariableValue, bInit, (flags AND VisuElems.Visu_InputFlags.Password) = 1, 'd'); ELSE VisuDlg_CheckedAppend(stOutputValue, stVariableValue, bInit, (flags AND VisuElems.Visu_InputFlags.Password) = 1, 'D'); END_IF, VisuElemId=-1
    hotkey HotkeyInput Id=481116028928, Key=KeyDown=True, KeyName=F, ActionToExecute=Action=STSnippet=IF bShift THEN VisuDlg_CheckedAppend(stOutputValue, stVariableValue, bInit, (flags AND VisuElems.Visu_InputFlags.Password) = 1, 'f'); ELSE VisuDlg_CheckedAppend(stOutputValue, stVariableValue, bInit, (flags AND VisuElems.Visu_InputFlags.Password) = 1, 'F'); END_IF, VisuElemId=-1
    hotkey HotkeyInput Id=481117077504, Key=KeyDown=True, KeyName=G, ActionToExecute=Action=STSnippet=IF bShift THEN VisuDlg_CheckedAppend(stOutputValue, stVariableValue, bInit, (flags AND VisuElems.Visu_InputFlags.Password) = 1, 'g'); ELSE VisuDlg_CheckedAppend(stOutputValue, stVariableValue, bInit, (flags AND VisuElems.Visu_InputFlags.Password) = 1, 'G'); END_IF, VisuElemId=-1
    hotkey HotkeyInput Id=481118126080, Key=KeyDown=True, KeyName=H, ActionToExecute=Action=STSnippet=IF bShift THEN VisuDlg_CheckedAppend(stOutputValue, stVariableValue, bInit, (flags AND VisuElems.Visu_InputFlags.Password) = 1, 'h'); ELSE VisuDlg_CheckedAppend(stOutputValue, stVariableValue, bInit, (flags AND VisuElems.Visu_InputFlags.Password) = 1, 'H'); END_IF, VisuElemId=-1
    hotkey HotkeyInput Id=481119174656, Key=KeyDown=True, KeyName=J, ActionToExecute=Action=STSnippet=IF bShift THEN VisuDlg_CheckedAppend(stOutputValue, stVariableValue, bInit, (flags AND VisuElems.Visu_InputFlags.Password) = 1, 'j'); ELSE VisuDlg_CheckedAppend(stOutputValue, stVariableValue, bInit, (flags AND VisuElems.Visu_InputFlags.Password) = 1, 'J'); END_IF, VisuElemId=-1
    hotkey HotkeyInput Id=481120223232, Key=KeyDown=True, KeyName=K, ActionToExecute=Action=STSnippet=IF bShift THEN VisuDlg_CheckedAppend(stOutputValue, stVariableValue, bInit, (flags AND VisuElems.Visu_InputFlags.Password) = 1, 'k'); ELSE VisuDlg_CheckedAppend(stOutputValue, stVariableValue, bInit, (flags AND VisuElems.Visu_InputFlags.Password) = 1, 'K'); END_IF, VisuElemId=-1
    hotkey HotkeyInput Id=481121271808, Key=KeyDown=True, KeyName=L, ActionToExecute=Action=STSnippet=IF bShift THEN VisuDlg_CheckedAppend(stOutputValue, stVariableValue, bInit, (flags AND VisuElems.Visu_InputFlags.Password) = 1, 'l'); ELSE VisuDlg_CheckedAppend(stOutputValue, stVariableValue, bInit, (flags AND VisuElems.Visu_InputFlags.Password) = 1, 'L'); END_IF, VisuElemId=-1
    hotkey HotkeyInput Id=481122320384, Key=KeyDown=True, KeyName=Z, ActionToExecute=Action=STSnippet=IF bShift THEN VisuDlg_CheckedAppend(stOutputValue, stVariableValue, bInit, (flags AND VisuElems.Visu_InputFlags.Password) = 1, 'z'); ELSE VisuDlg_CheckedAppend(stOutputValue, stVariableValue, bInit, (flags AND VisuElems.Visu_InputFlags.Password) = 1, 'Z'); END_IF, VisuElemId=-1
    hotkey HotkeyInput Id=481123368960, Key=KeyDown=True, KeyName=X, ActionToExecute=Action=STSnippet=IF bShift THEN VisuDlg_CheckedAppend(stOutputValue, stVariableValue, bInit, (flags AND VisuElems.Visu_InputFlags.Password) = 1, 'x'); ELSE VisuDlg_CheckedAppend(stOutputValue, stVariableValue, bInit, (flags AND VisuElems.Visu_InputFlags.Password) = 1, 'X'); END_IF, VisuElemId=-1
    hotkey HotkeyInput Id=481124417536, Key=KeyDown=True, KeyName=C, ActionToExecute=Action=STSnippet=IF bShift THEN VisuDlg_CheckedAppend(stOutputValue, stVariableValue, bInit, (flags AND VisuElems.Visu_InputFlags.Password) = 1, 'c'); ELSE VisuDlg_CheckedAppend(stOutputValue, stVariableValue, bInit, (flags AND VisuElems.Visu_InputFlags.Password) = 1, 'C'); END_IF, VisuElemId=-1
    hotkey HotkeyInput Id=481125466112, Key=KeyDown=True, KeyName=V, ActionToExecute=Action=STSnippet=IF bShift THEN VisuDlg_CheckedAppend(stOutputValue, stVariableValue, bInit, (flags AND VisuElems.Visu_InputFlags.Password) = 1, 'v'); ELSE VisuDlg_CheckedAppend(stOutputValue, stVariableValue, bInit, (flags AND VisuElems.Visu_InputFlags.Password) = 1, 'V'); END_IF, VisuElemId=-1
    hotkey HotkeyInput Id=481126514688, Key=KeyDown=True, KeyName=B, ActionToExecute=Action=STSnippet=IF bShift THEN VisuDlg_CheckedAppend(stOutputValue, stVariableValue, bInit, (flags AND VisuElems.Visu_InputFlags.Password) = 1, 'b'); ELSE VisuDlg_CheckedAppend(stOutputValue, stVariableValue, bInit, (flags AND VisuElems.Visu_InputFlags.Password) = 1, 'B'); END_IF, VisuElemId=-1
    hotkey HotkeyInput Id=481127563264, Key=KeyDown=True, KeyName=N, ActionToExecute=Action=STSnippet=IF bShift THEN VisuDlg_CheckedAppend(stOutputValue, stVariableValue, bInit, (flags AND VisuElems.Visu_InputFlags.Password) = 1, 'n'); ELSE VisuDlg_CheckedAppend(stOutputValue, stVariableValue, bInit, (flags AND VisuElems.Visu_InputFlags.Password) = 1, 'N'); END_IF, VisuElemId=-1
    hotkey HotkeyInput Id=481128611840, Key=KeyDown=True, KeyName=M, ActionToExecute=Action=STSnippet=IF bShift THEN VisuDlg_CheckedAppend(stOutputValue, stVariableValue, bInit, (flags AND VisuElems.Visu_InputFlags.Password) = 1, 'm'); ELSE VisuDlg_CheckedAppend(stOutputValue, stVariableValue, bInit, (flags AND VisuElems.Visu_InputFlags.Password) = 1, 'M'); END_IF, VisuElemId=-1
    hotkey HotkeyInput Id=481129660416, Key=KeyDown=True, KeyName=COMMA, ActionToExecute=Action=STSnippet=IF bShift THEN VisuDlg_CheckedAppend(stOutputValue, stVariableValue, bInit, (flags AND VisuElems.Visu_InputFlags.Password) = 1, ','); ELSE VisuDlg_CheckedAppend(stOutputValue, stVariableValue, bInit, (flags AND VisuElems.Visu_InputFlags.Password) = 1, '.'); END_IF, VisuElemId=-1
    hotkey HotkeyInput Id=481131757568, Key=KeyDown=True, KeyName=NUM1, ActionToExecute=Action=STSnippet=VisuDlg_CheckedAppend(stOutputValue, stVariableValue, bInit, (flags AND VisuElems.Visu_InputFlags.Password) = 1, '1');, VisuElemId=-1
    hotkey HotkeyInput Id=481132806144, Key=KeyDown=True, KeyName=NUM2, ActionToExecute=Action=STSnippet=VisuDlg_CheckedAppend(stOutputValue, stVariableValue, bInit, (flags AND VisuElems.Visu_InputFlags.Password) = 1, '2');, VisuElemId=-1
    hotkey HotkeyInput Id=481133854720, Key=KeyDown=True, KeyName=NUM3, ActionToExecute=Action=STSnippet=VisuDlg_CheckedAppend(stOutputValue, stVariableValue, bInit, (flags AND VisuElems.Visu_InputFlags.Password) = 1, '3');, VisuElemId=-1
    hotkey HotkeyInput Id=481134903296, Key=KeyDown=True, KeyName=NUM4, ActionToExecute=Action=STSnippet=VisuDlg_CheckedAppend(stOutputValue, stVariableValue, bInit, (flags AND VisuElems.Visu_InputFlags.Password) = 1, '4');, VisuElemId=-1
    hotkey HotkeyInput Id=481135951872, Key=KeyDown=True, KeyName=NUM5, ActionToExecute=Action=STSnippet=VisuDlg_CheckedAppend(stOutputValue, stVariableValue, bInit, (flags AND VisuElems.Visu_InputFlags.Password) = 1, '5');, VisuElemId=-1
    hotkey HotkeyInput Id=481137000448, Key=KeyDown=True, KeyName=NUM6, ActionToExecute=Action=STSnippet=VisuDlg_CheckedAppend(stOutputValue, stVariableValue, bInit, (flags AND VisuElems.Visu_InputFlags.Password) = 1, '6');, VisuElemId=-1
    hotkey HotkeyInput Id=481138049024, Key=KeyDown=True, KeyName=NUM7, ActionToExecute=Action=STSnippet=VisuDlg_CheckedAppend(stOutputValue, stVariableValue, bInit, (flags AND VisuElems.Visu_InputFlags.Password) = 1, '7');, VisuElemId=-1
    hotkey HotkeyInput Id=481139097600, Key=KeyDown=True, KeyName=NUM8, ActionToExecute=Action=STSnippet=VisuDlg_CheckedAppend(stOutputValue, stVariableValue, bInit, (flags AND VisuElems.Visu_InputFlags.Password) = 1, '8');, VisuElemId=-1
    hotkey HotkeyInput Id=481140146176, Key=KeyDown=True, KeyName=NUM9, ActionToExecute=Action=STSnippet=VisuDlg_CheckedAppend(stOutputValue, stVariableValue, bInit, (flags AND VisuElems.Visu_InputFlags.Password) = 1, '9');, VisuElemId=-1
    hotkey HotkeyInput Id=481141194752, Key=KeyDown=True, KeyName=NUM0, ActionToExecute=Action=STSnippet=VisuDlg_CheckedAppend(stOutputValue, stVariableValue, bInit, (flags AND VisuElems.Visu_InputFlags.Password) = 1, '0');, VisuElemId=-1
END_VISUALIZATION

// ---- VISUs/Internal/Numpad.TcVIS
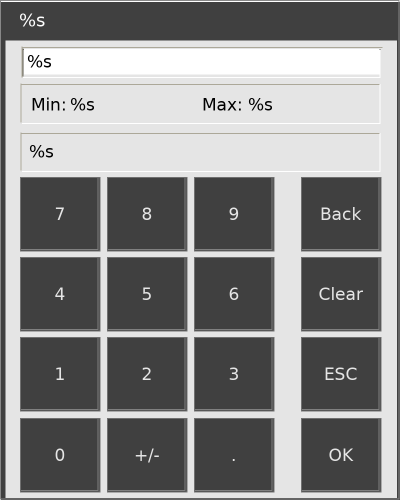
VISUALIZATION Numpad  // 400x500
VAR_INPUT
	stVariableValue 						: STRING;
	stMin 									: STRING;
	stMax 									: STRING;
	stTitle 								: STRING;
	flags 									: DWORD;
END_VAR
VAR
	bInit 									: BOOL;
	stMessage 								: STRING;
	stOutputValue 							: STRING;
END_VAR
    Rectangle (4,170 395x83)
    Rectangle (4,253 395x80)
    Rectangle (4,333 395x80)
    Rectangle (4,413 395x85)
    Button (301,418 80x74), "OK"
        OnMouseDown: CloseDialog Dialog=Numpad, Result=OK, NumpadKeypad=True, NumpadKeypadSet=True
    Button (301,337 80x74), "ESC"
        OnMouseDown: CloseDialog Dialog=Numpad, Result=Cancel, NumpadKeypad=True, NumpadKeypadSet=True
    Button (301,257 80x74), "Clear"
        OnMouseDown: execute {
            stVariableValue := '';
            stOutputValue := '';
            flags := flags AND 16#0008;
            flags := flags AND 16#0010;
        }
    Button (301,177 80x74), "Back"
        OnMouseDown: execute { VisuDlg_CheckedBack(stOutputValue, stVariableValue, bInit); }
    Button (194,418 80x74), "."
        OnMouseDown: execute { VisuDlg_CheckedAppend(stOutputValue, stVariableValue, bInit, (flags AND VisuElems.Visu_InputFlags.Password) = 1, '.'); }
    Button (107,418 80x74), "+/-"
        OnMouseDown: execute { VisuDlg_CheckedChangeSign(stOutputValue, stVariableValue, bInit, (flags AND VisuElems.Visu_InputFlags.Password) = 1); }
    Button (20,418 80x74), "0"
        OnMouseDown: execute { VisuDlg_CheckedAppend(stOutputValue, stVariableValue, bInit, (flags AND VisuElems.Visu_InputFlags.Password) = 1, '0'); }
    Button (20,337 80x74), "1"
        OnMouseDown: execute { VisuDlg_CheckedAppend(stOutputValue, stVariableValue, bInit, (flags AND VisuElems.Visu_InputFlags.Password) = 1, '1'); }
    Button (107,337 80x74), "2"
        OnMouseDown: execute { VisuDlg_CheckedAppend(stOutputValue, stVariableValue, bInit, (flags AND VisuElems.Visu_InputFlags.Password) = 1, '2'); }
    Button (194,337 80x74), "3"
        OnMouseDown: execute { VisuDlg_CheckedAppend(stOutputValue, stVariableValue, bInit, (flags AND VisuElems.Visu_InputFlags.Password) = 1, '3'); }
    Button (20,257 80x74), "4"
        OnMouseDown: execute { VisuDlg_CheckedAppend(stOutputValue, stVariableValue, bInit, (flags AND VisuElems.Visu_InputFlags.Password) = 1, '4'); }
    Button (107,257 80x74), "5"
        OnMouseDown: execute { VisuDlg_CheckedAppend(stOutputValue, stVariableValue, bInit, (flags AND VisuElems.Visu_InputFlags.Password) = 1, '5'); }
    Button (194,257 80x74), "6"
        OnMouseDown: execute { VisuDlg_CheckedAppend(stOutputValue, stVariableValue, bInit, (flags AND VisuElems.Visu_InputFlags.Password) = 1, '6'); }
    Button (20,177 80x74), "7"
        OnMouseDown: execute { VisuDlg_CheckedAppend(stOutputValue, stVariableValue, bInit, (flags AND VisuElems.Visu_InputFlags.Password) = 1, '7'); }
    Button (107,177 80x74), "8"
        OnMouseDown: execute { VisuDlg_CheckedAppend(stOutputValue, stVariableValue, bInit, (flags AND VisuElems.Visu_InputFlags.Password) = 1, '8'); }
    Button (194,177 80x74), "9"
        OnMouseDown: execute { VisuDlg_CheckedAppend(stOutputValue, stVariableValue, bInit, (flags AND VisuElems.Visu_InputFlags.Password) = 1, '9'); }
    Rectangle (4,38 393x48)
    Rectangle (4,85 393x85)
    Rectangle (67,92 127x25), "%s", text variable: stMin, invisible if: LEN(stMin) = 0
    Rectangle (245,92 127x25), "%s", text variable: stMax, invisible if: LEN(stMax) = 0
    Rectangle (199,92 45x25), "Max:", text variable: stMin, invisible if: LEN(stMax) = 0
        p55702900: SEL(((UDINT_TO_DINT(flags AND 16#0010))=16#0010),16#FF000000,16#FFFF0000)
    Rectangle (396,498 4x4)
    Rectangle (397,2 4x500)
    Rectangle (1,3 4x499)
    Rectangle (1,2 399x38)
    Rectangle (16,8 375x25), "%s", text variable: stTitle
    Rectangle (1,498 400x4)
    Polyline (21,122) (21,84) (379,84)
    Polyline (21,170) (21,133) (379,133)
    Polyline (22,77) (22,47) (382,47)
    Polyline (22,171) (380,171) (380,133)
    Polyline (22,123) (380,123) (380,84)
    Polyline (23,77) (380,77) (380,49)
    Polyline (23,76) (23,49) (380,49)
    Rectangle (26,139 349x25), "%s", text variable: stMessage
    Rectangle (28,92 41x25), "Min:", text variable: stMin, invisible if: LEN(stMin) = 0
        p55702900: SEL(((UDINT_TO_DINT(flags AND 16#0008))=16#0008),16#FF000000,16#FFFF0000)
    Rectangle (24,49 355x25), "%s", text variable: stOutputValue
    hotkey HotkeyInput Id=481049968640, Key=KeyDown=True, KeyName=0, ActionToExecute=Action=STSnippet=VisuDlg_CheckedAppend(stOutputValue, stVariableValue, bInit, (flags AND VisuElems.Visu_InputFlags.Password) = 1, '0');, VisuElemId=-1
    hotkey HotkeyInput Id=481053114368, Key=KeyDown=True, KeyName=NUM0, ActionToExecute=Action=STSnippet=VisuDlg_CheckedAppend(stOutputValue, stVariableValue, bInit, (flags AND VisuElems.Visu_InputFlags.Password) = 1, '0');, VisuElemId=-1
    hotkey HotkeyInput Id=481054162944, Key=KeyDown=True, KeyName=1, ActionToExecute=Action=STSnippet=VisuDlg_CheckedAppend(stOutputValue, stVariableValue, bInit, (flags AND VisuElems.Visu_InputFlags.Password) = 1, '1');, VisuElemId=-1
    hotkey HotkeyInput Id=481055211520, Key=KeyDown=True, KeyName=NUM1, ActionToExecute=Action=STSnippet=VisuDlg_CheckedAppend(stOutputValue, stVariableValue, bInit, (flags AND VisuElems.Visu_InputFlags.Password) = 1, '1');, VisuElemId=-1
    hotkey HotkeyInput Id=481056260096, Key=KeyDown=True, KeyName=2, ActionToExecute=Action=STSnippet=VisuDlg_CheckedAppend(stOutputValue, stVariableValue, bInit, (flags AND VisuElems.Visu_InputFlags.Password) = 1, '2');, VisuElemId=-1
    hotkey HotkeyInput Id=481057308672, Key=KeyDown=True, KeyName=NUM2, ActionToExecute=Action=STSnippet=VisuDlg_CheckedAppend(stOutputValue, stVariableValue, bInit, (flags AND VisuElems.Visu_InputFlags.Password) = 1, '2');, VisuElemId=-1
    hotkey HotkeyInput Id=481058357248, Key=KeyDown=True, KeyName=3, ActionToExecute=Action=STSnippet=VisuDlg_CheckedAppend(stOutputValue, stVariableValue, bInit, (flags AND VisuElems.Visu_InputFlags.Password) = 1, '3');, VisuElemId=-1
    hotkey HotkeyInput Id=481059405824, Key=KeyDown=True, KeyName=NUM3, ActionToExecute=Action=STSnippet=VisuDlg_CheckedAppend(stOutputValue, stVariableValue, bInit, (flags AND VisuElems.Visu_InputFlags.Password) = 1, '3');, VisuElemId=-1
    hotkey HotkeyInput Id=481060454400, Key=KeyDown=True, KeyName=4, ActionToExecute=Action=STSnippet=VisuDlg_CheckedAppend(stOutputValue, stVariableValue, bInit, (flags AND VisuElems.Visu_InputFlags.Password) = 1, '4');, VisuElemId=-1
    hotkey HotkeyInput Id=481061502976, Key=KeyDown=True, KeyName=NUM4, ActionToExecute=Action=STSnippet=VisuDlg_CheckedAppend(stOutputValue, stVariableValue, bInit, (flags AND VisuElems.Visu_InputFlags.Password) = 1, '4');, VisuElemId=-1
    hotkey HotkeyInput Id=481062551552, Key=KeyDown=True, KeyName=5, ActionToExecute=Action=STSnippet=VisuDlg_CheckedAppend(stOutputValue, stVariableValue, bInit, (flags AND VisuElems.Visu_InputFlags.Password) = 1, '5');, VisuElemId=-1
    hotkey HotkeyInput Id=481063600128, Key=KeyDown=True, KeyName=NUM5, ActionToExecute=Action=STSnippet=VisuDlg_CheckedAppend(stOutputValue, stVariableValue, bInit, (flags AND VisuElems.Visu_InputFlags.Password) = 1, '5');, VisuElemId=-1
    hotkey HotkeyInput Id=481064648704, Key=KeyDown=True, KeyName=6, ActionToExecute=Action=STSnippet=VisuDlg_CheckedAppend(stOutputValue, stVariableValue, bInit, (flags AND VisuElems.Visu_InputFlags.Password) = 1, '6');, VisuElemId=-1
    hotkey HotkeyInput Id=481065697280, Key=KeyDown=True, KeyName=NUM6, ActionToExecute=Action=STSnippet=VisuDlg_CheckedAppend(stOutputValue, stVariableValue, bInit, (flags AND VisuElems.Visu_InputFlags.Password) = 1, '6');, VisuElemId=-1
    hotkey HotkeyInput Id=481066745856, Key=KeyDown=True, KeyName=7, ActionToExecute=Action=STSnippet=VisuDlg_CheckedAppend(stOutputValue, stVariableValue, bInit, (flags AND VisuElems.Visu_InputFlags.Password) = 1, '7');, VisuElemId=-1
    hotkey HotkeyInput Id=481067794432, Key=KeyDown=True, KeyName=NUM7, ActionToExecute=Action=STSnippet=VisuDlg_CheckedAppend(stOutputValue, stVariableValue, bInit, (flags AND VisuElems.Visu_InputFlags.Password) = 1, '7');, VisuElemId=-1
    hotkey HotkeyInput Id=481068843008, Key=KeyDown=True, KeyName=8, ActionToExecute=Action=STSnippet=VisuDlg_CheckedAppend(stOutputValue, stVariableValue, bInit, (flags AND VisuElems.Visu_InputFlags.Password) = 1, '8');, VisuElemId=-1
    hotkey HotkeyInput Id=481069891584, Key=KeyDown=True, KeyName=NUM8, ActionToExecute=Action=STSnippet=VisuDlg_CheckedAppend(stOutputValue, stVariableValue, bInit, (flags AND VisuElems.Visu_InputFlags.Password) = 1, '8');, VisuElemId=-1
    hotkey HotkeyInput Id=481070940160, Key=KeyDown=True, KeyName=9, ActionToExecute=Action=STSnippet=VisuDlg_CheckedAppend(stOutputValue, stVariableValue, bInit, (flags AND VisuElems.Visu_InputFlags.Password) = 1, '9');, VisuElemId=-1
    hotkey HotkeyInput Id=481071988736, Key=KeyDown=True, KeyName=NUM9, ActionToExecute=Action=STSnippet=VisuDlg_CheckedAppend(stOutputValue, stVariableValue, bInit, (flags AND VisuElems.Visu_InputFlags.Password) = 1, '9');, VisuElemId=-1
    hotkey HotkeyInput Id=481073037312, Key=KeyDown=True, KeyName=SUBTRACT, ActionToExecute=Action=STSnippet=VisuDlg_CheckedChangeSign(stOutputValue, stVariableValue, bInit, (flags AND VisuElems.Visu_InputFlags.Password) = 1);, VisuElemId=-1
    hotkey HotkeyInput Id=481074085888, Key=KeyDown=True, KeyName=COMMA, ActionToExecute=Action=STSnippet=VisuDlg_CheckedAppend(stOutputValue, stVariableValue, bInit, (flags AND VisuElems.Visu_InputFlags.Password) = 1, '.');, VisuElemId=-1
    hotkey HotkeyInput Id=481075134464, Key=KeyDown=True, KeyName=BACKSPACE, ActionToExecute=Action=STSnippet=VisuDlg_CheckedBack(stOutputValue, stVariableValue, bInit);, VisuElemId=-1
    hotkey HotkeyInput Id=481076183040, Key=KeyDown=True, KeyName=DELETE, ActionToExecute=Action=STSnippet=stVariableValue := ''; stOutputValue := ''; flags := flags AND 16#0008; flags := flags AND 16#0010;, VisuElemId=-1
    hotkey HotkeyInput Id=481077231616, Key=KeyDown=True, KeyName=ESCAPE, ActionToExecute=Action=Dialog=Numpad, Result=Cancel, NumpadKeypad=True, NumpadKeypadSet=True, VisuElemId=-1
    hotkey HotkeyInput Id=481078280192, Key=KeyDown=True, KeyName=RETURN_KEY, ActionToExecute=Action=Dialog=Numpad, Result=OK, NumpadKeypad=True, NumpadKeypadSet=True, VisuElemId=-1
END_VISUALIZATION

// ---- VISUs/Internal/PH_Bottom.TcVIS
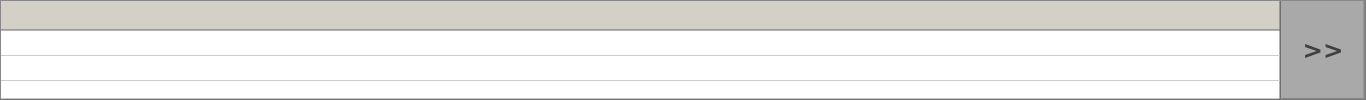
VISUALIZATION PH_Bottom  // 1366x100
VAR_IN_OUT
	bReset 									: BOOL;
	arrEventVisu							: ARRAY [1..GVL_EHS.diNoOfEvents] OF ST_EventHistoricalSimple;	 
END_VAR
    Table (0,0 1280x100), data array: GVL_EHS.arrEventVisu
        p3854506369: GVL_EHS.arrEventVisu[INDEX].dwID
        p505689113: Date End
        p1218418051: GVL_EHS.arrEventVisu[INDEX].dtDateEnd
        p2237128397: Date Begin
        p3723444502: GVL_EHS.arrEventVisu[INDEX].dtDateBegin
        p4092479075: Param
        p2170511999: GVL_EHS.arrEventVisu[INDEX].dwParam
        p511219082: Class
        p1892666644: GVL_EHS.arrEventVisu[INDEX].dwClass
        p1755163831: Message
        p338671338: GVL_EHS.arrEventVisu[INDEX].wsMessage
        Columns.Column.[2].Template: GVL_EHS.arrEventVisu[INDEX].dwColor
        Columns.Column.[0].Template: GVL_EHS.arrEventVisu[INDEX].dwColor
        Columns.Column.[1].Template: GVL_EHS.arrEventVisu[INDEX].dwColor
        Columns.Column.[4].Template: GVL_EHS.arrEventVisu[INDEX].dwColor
        Columns.Column.[3].Template: GVL_EHS.arrEventVisu[INDEX].dwColor
        Columns.Column.[5].Template: GVL_EHS.arrEventVisu[INDEX].dwColor
    Button (1280,0 86x100), ">>"
        OnMouseDown: execute { GVL_HMI.iFrameNumber:=1; GVL_HMI.bMenu:=FALSE; }
END_VISUALIZATION

// ---- VISUs/Internal/PH_ControllerInfo.TcVIS
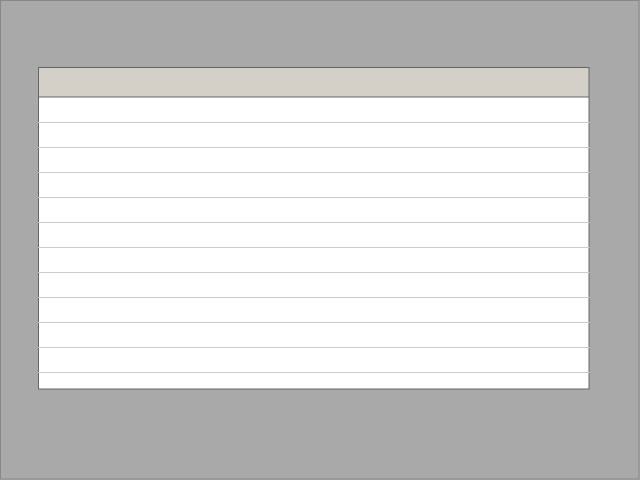
VISUALIZATION PH_ControllerInfo  // 640x480
VAR_IN_OUT
	strTargetType							: STRING(20);
	strHardwareModel						: STRING(10);
	strHardwareSerialNo						: STRING(12);
	strHardwareVersion						: STRING(4);
	strHardwareDate							: STRING(10);
	strHardwareCPU							: STRING(10);
	strImageDevice							: STRING(20);
	strImageVersion							: STRING(10);
	strImageLevel							: STRING(10);
	strImageOsName							: STRING(20);
	strImageOsVersion						: STRING(8);
	strTwinCATVersion						: STRING(4);
	strTwinCATRevision						: STRING(4);
	strTwinCATBuild							: STRING(8);
	strTwinCATLevel							: STRING(20);
	strAmsNetId								: STRING(23);
	arrDevIdent								: ARRAY [0..1, 1..16] OF STRING(23) ;
	wDeviceInfo								: WORD;
	iSelectedRow							: INT;
END_VAR
    Table (38,67 551x322), data array: arrDevIdent
        p338671338: MAIN.fbAutostartVisu.stDevIdent.strHardwareSerialNo
        p2170511999: MAIN.fbAutostartVisu.stDevIdent.strHardwareVersion
        p3723444502: MAIN.fbAutostartVisu.stDevIdent.strHardwareDate
        p1218418051: MAIN.fbAutostartVisu.stDevIdent.strHardwareCPU
        p746581629: MAIN.fbAutostartVisu.stDevIdent.strImageDevice
        p3104783080: MAIN.fbAutostartVisu.stDevIdent.strImageVersion
        p2501879983: MAIN.fbAutostartVisu.stDevIdent.strImageLevel
        p7306298: MAIN.fbAutostartVisu.stDevIdent.strImageOsName
        p1933151965: MAIN.fbAutostartVisu.stDevIdent.strImageOsVersion
        p3863566920: MAIN.fbAutostartVisu.stDevIdent.strTwinCATVersion
        p2192122294: MAIN.fbAutostartVisu.stDevIdent.strTwinCATRevision
        p400160035: MAIN.fbAutostartVisu.stDevIdent.strTwinCATBuild
        p1265227338: MAIN.fbAutostartVisu.stDevIdent.strTwinCATLevel
        p3726181087: MAIN.fbAutostartVisu.stDevIdent.strAmsNetId
        p3854506369: arrDevIdent[0,INDEX]
        p1892666644: arrDevIdent[1,INDEX]
        p1137915858: iSelectedRow
END_VISUALIZATION

